REGION Network 68: **** 4.4 - Machine Status - Calculation **** Que Message Request 13 / **** 4.4 - Machine Status - Calculation **** Queue Message Request 13
   // Que Message Request 13 / Queue Message Request 13
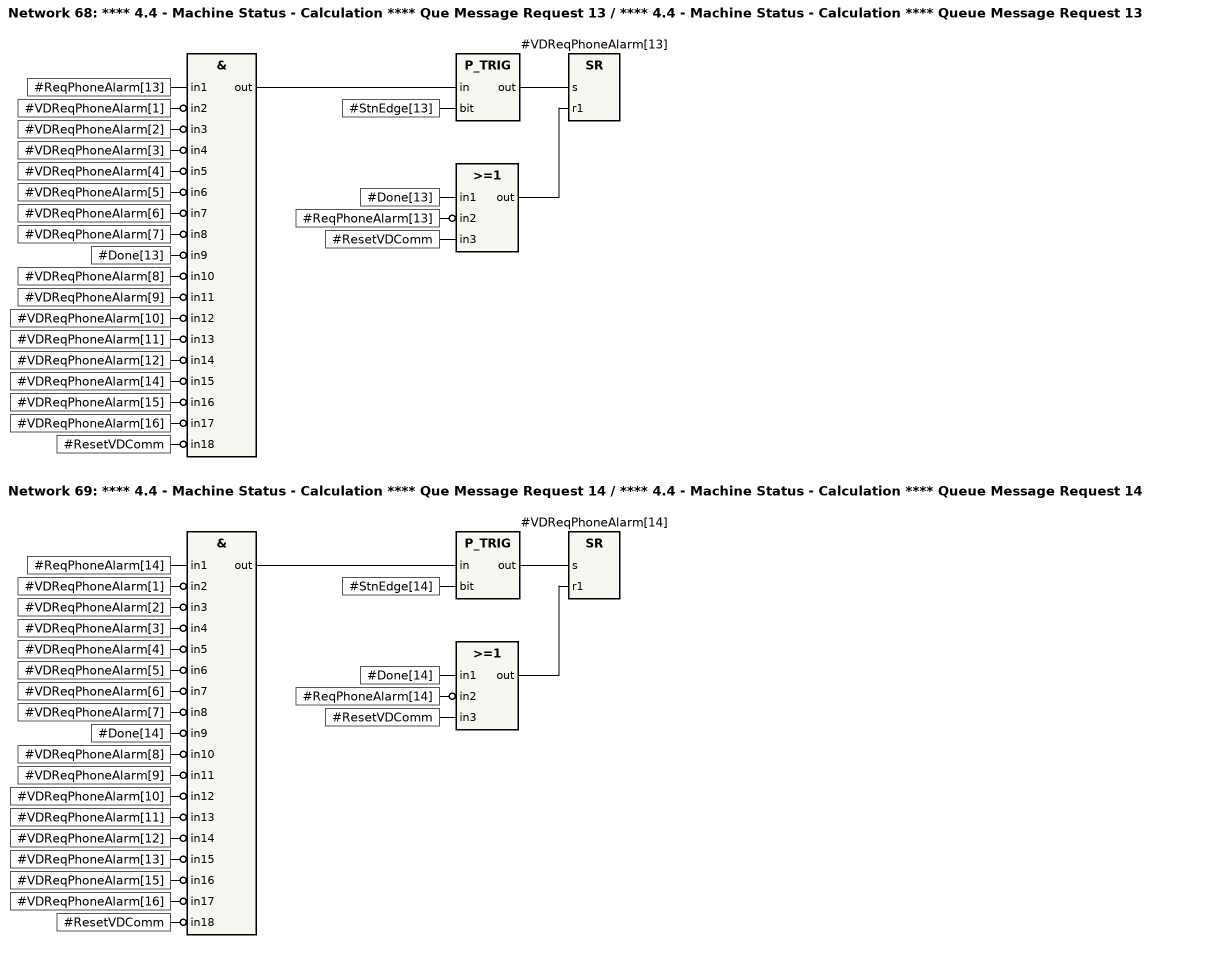
   #_w1 := #ReqPhoneAlarm[13] AND NOT #VDReqPhoneAlarm[1] AND NOT #VDReqPhoneAlarm[2] AND NOT #VDReqPhoneAlarm[3] AND NOT #VDReqPhoneAlarm[4] AND NOT #VDReqPhoneAlarm[5] AND NOT #VDReqPhoneAlarm[6] AND NOT #VDReqPhoneAlarm[7] AND NOT #Done[13] AND NOT #VDReqPhoneAlarm[8] AND NOT #VDReqPhoneAlarm[9] AND NOT #VDReqPhoneAlarm[10] AND NOT #VDReqPhoneAlarm[11] AND NOT #VDReqPhoneAlarm[12] AND NOT #VDReqPhoneAlarm[14] AND NOT #VDReqPhoneAlarm[15] AND NOT #VDReqPhoneAlarm[16] AND NOT #ResetVDComm;
   #_w2 := #_w1 AND NOT #StnEdge[13];   // rising edge
   #StnEdge[13] := #_w1;
   IF #_w2 THEN
       #VDReqPhoneAlarm[13] := TRUE;   // SR flip-flop
   END_IF;
   IF #Done[13] OR NOT #ReqPhoneAlarm[13] OR #ResetVDComm THEN #VDReqPhoneAlarm[13] := FALSE; END_IF;
END_REGION

REGION Network 69: **** 4.4 - Machine Status - Calculation **** Que Message Request 14 / **** 4.4 - Machine Status - Calculation **** Queue Message Request 14
   // Que Message Request 14 / Queue Message Request 14
   #_w1 := #ReqPhoneAlarm[14] AND NOT #VDReqPhoneAlarm[1] AND NOT #VDReqPhoneAlarm[2] AND NOT #VDReqPhoneAlarm[3] AND NOT #VDReqPhoneAlarm[4] AND NOT #VDReqPhoneAlarm[5] AND NOT #VDReqPhoneAlarm[6] AND NOT #VDReqPhoneAlarm[7] AND NOT #Done[14] AND NOT #VDReqPhoneAlarm[8] AND NOT #VDReqPhoneAlarm[9] AND NOT #VDReqPhoneAlarm[10] AND NOT #VDReqPhoneAlarm[11] AND NOT #VDReqPhoneAlarm[12] AND NOT #VDReqPhoneAlarm[13] AND NOT #VDReqPhoneAlarm[15] AND NOT #VDReqPhoneAlarm[16] AND NOT #ResetVDComm;
   #_w2 := #_w1 AND NOT #StnEdge[14];   // rising edge
   #StnEdge[14] := #_w1;
   IF #_w2 THEN
       #VDReqPhoneAlarm[14] := TRUE;   // SR flip-flop
   END_IF;
   IF #Done[14] OR NOT #ReqPhoneAlarm[14] OR #ResetVDComm THEN #VDReqPhoneAlarm[14] := FALSE; END_IF;
END_REGION

REGION Network 70: **** 4.4 - Machine Status - Calculation **** Que Message Request 15 / **** 4.4 - Machine Status - Calculation **** Queue Message Request 15
   // Que Message Request 15 / Queue Message Request 15
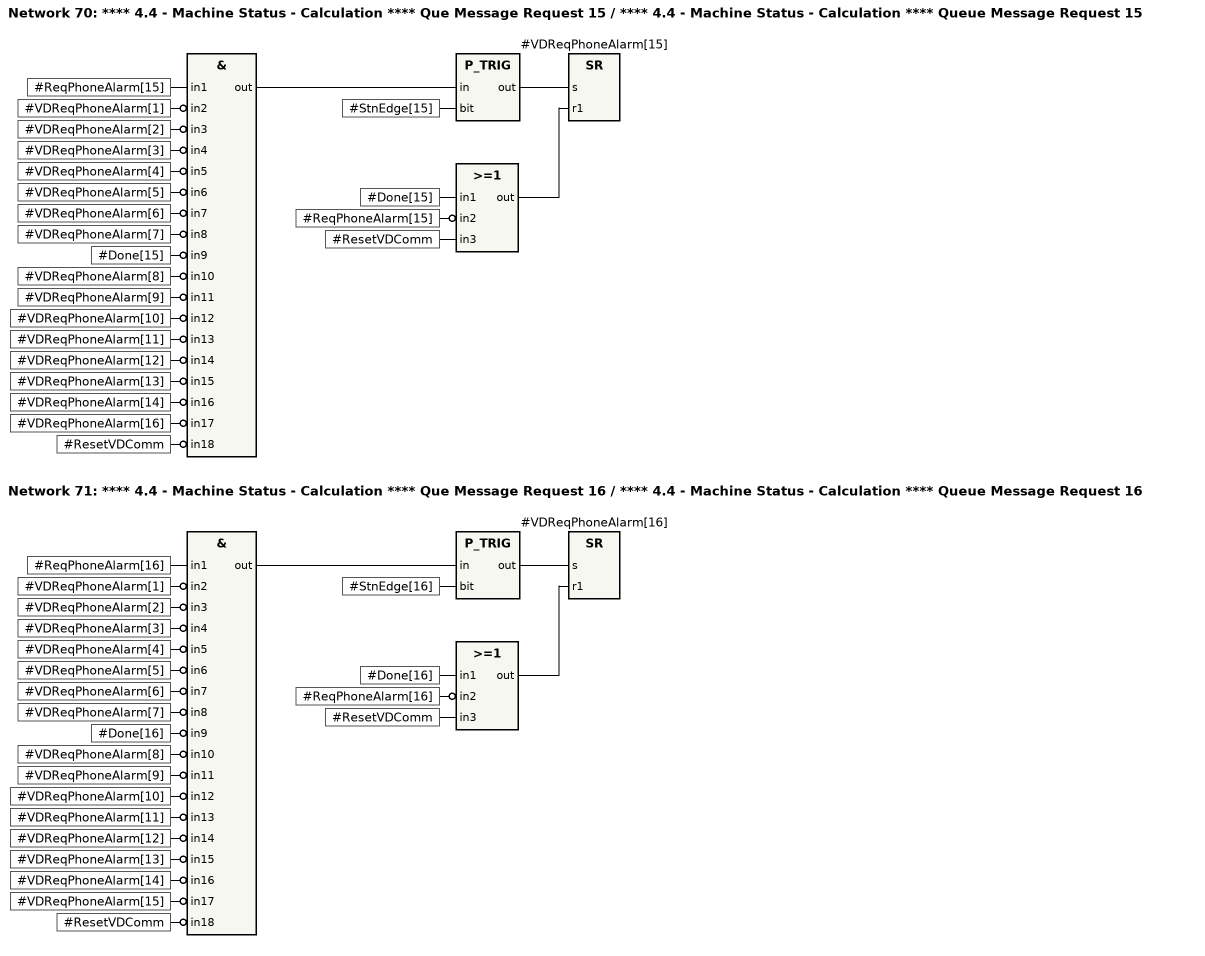
   #_w1 := #ReqPhoneAlarm[15] AND NOT #VDReqPhoneAlarm[1] AND NOT #VDReqPhoneAlarm[2] AND NOT #VDReqPhoneAlarm[3] AND NOT #VDReqPhoneAlarm[4] AND NOT #VDReqPhoneAlarm[5] AND NOT #VDReqPhoneAlarm[6] AND NOT #VDReqPhoneAlarm[7] AND NOT #Done[15] AND NOT #VDReqPhoneAlarm[8] AND NOT #VDReqPhoneAlarm[9] AND NOT #VDReqPhoneAlarm[10] AND NOT #VDReqPhoneAlarm[11] AND NOT #VDReqPhoneAlarm[12] AND NOT #VDReqPhoneAlarm[13] AND NOT #VDReqPhoneAlarm[14] AND NOT #VDReqPhoneAlarm[16] AND NOT #ResetVDComm;
   #_w2 := #_w1 AND NOT #StnEdge[15];   // rising edge
   #StnEdge[15] := #_w1;
   IF #_w2 THEN
       #VDReqPhoneAlarm[15] := TRUE;   // SR flip-flop
   END_IF;
   IF #Done[15] OR NOT #ReqPhoneAlarm[15] OR #ResetVDComm THEN #VDReqPhoneAlarm[15] := FALSE; END_IF;
END_REGION

REGION Network 71: **** 4.4 - Machine Status - Calculation **** Que Message Request 16 / **** 4.4 - Machine Status - Calculation **** Queue Message Request 16
   // Que Message Request 16 / Queue Message Request 16
   #_w1 := #ReqPhoneAlarm[16] AND NOT #VDReqPhoneAlarm[1] AND NOT #VDReqPhoneAlarm[2] AND NOT #VDReqPhoneAlarm[3] AND NOT #VDReqPhoneAlarm[4] AND NOT #VDReqPhoneAlarm[5] AND NOT #VDReqPhoneAlarm[6] AND NOT #VDReqPhoneAlarm[7] AND NOT #Done[16] AND NOT #VDReqPhoneAlarm[8] AND NOT #VDReqPhoneAlarm[9] AND NOT #VDReqPhoneAlarm[10] AND NOT #VDReqPhoneAlarm[11] AND NOT #VDReqPhoneAlarm[12] AND NOT #VDReqPhoneAlarm[13] AND NOT #VDReqPhoneAlarm[14] AND NOT #VDReqPhoneAlarm[15] AND NOT #ResetVDComm;
   #_w2 := #_w1 AND NOT #StnEdge[16];   // rising edge
   #StnEdge[16] := #_w1;
   IF #_w2 THEN
       #VDReqPhoneAlarm[16] := TRUE;   // SR flip-flop
   END_IF;
   IF #Done[16] OR NOT #ReqPhoneAlarm[16] OR #ResetVDComm THEN #VDReqPhoneAlarm[16] := FALSE; END_IF;
END_REGION

REGION Network 72: **** 4.6 - Machine status - Indication **** Animation / **** 4.6 - Machine status - Indication **** Animation SP1
   // Animation
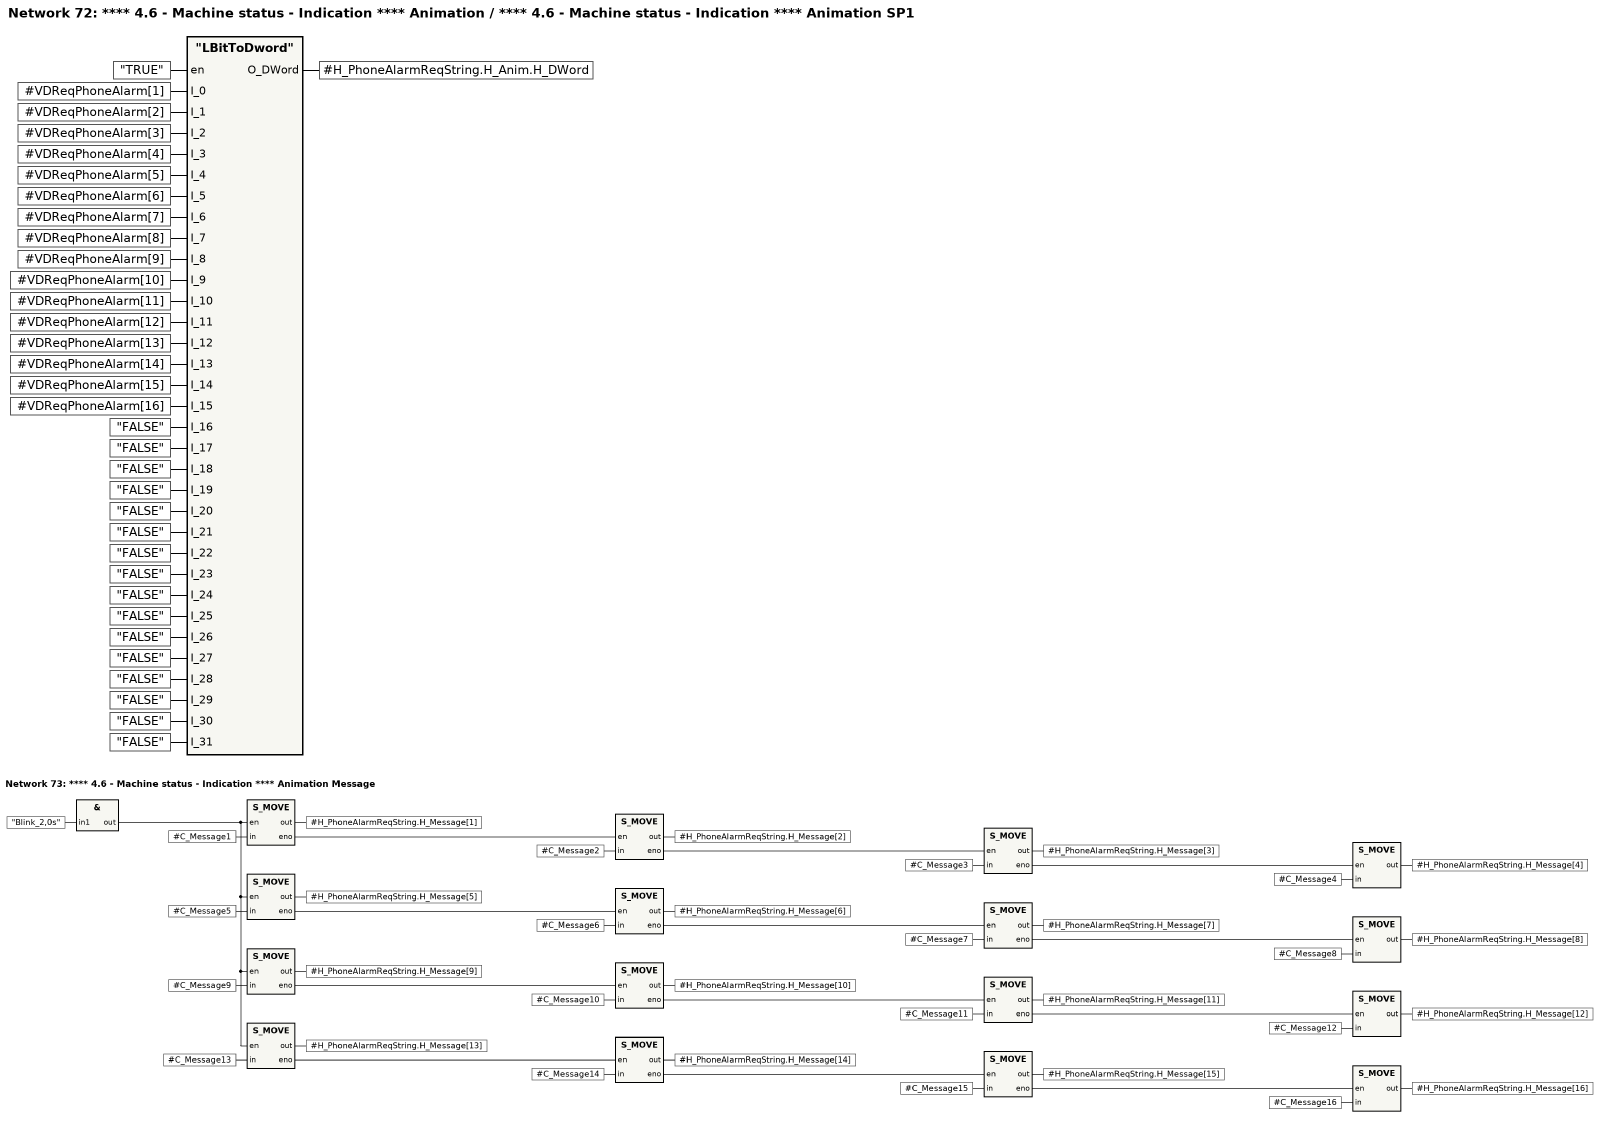
   IF "TRUE" THEN
       "LBitToDword"(I_0 := #VDReqPhoneAlarm[1],
                     I_1 := #VDReqPhoneAlarm[2],
                     I_2 := #VDReqPhoneAlarm[3],
                     I_3 := #VDReqPhoneAlarm[4],
                     I_4 := #VDReqPhoneAlarm[5],
                     I_5 := #VDReqPhoneAlarm[6],
                     I_6 := #VDReqPhoneAlarm[7],
                     I_7 := #VDReqPhoneAlarm[8],
                     I_8 := #VDReqPhoneAlarm[9],
                     I_9 := #VDReqPhoneAlarm[10],
                     I_10 := #VDReqPhoneAlarm[11],
                     I_11 := #VDReqPhoneAlarm[12],
                     I_12 := #VDReqPhoneAlarm[13],
                     I_13 := #VDReqPhoneAlarm[14],
                     I_14 := #VDReqPhoneAlarm[15],
                     I_15 := #VDReqPhoneAlarm[16],
                     I_16 := "FALSE",
                     I_17 := "FALSE",
                     I_18 := "FALSE",
                     I_19 := "FALSE",
                     I_20 := "FALSE",
                     I_21 := "FALSE",
                     I_22 := "FALSE",
                     I_23 := "FALSE",
                     I_24 := "FALSE",
                     I_25 := "FALSE",
                     I_26 := "FALSE",
                     I_27 := "FALSE",
                     I_28 := "FALSE",
                     I_29 := "FALSE",
                     I_30 := "FALSE",
                     I_31 := "FALSE",
                     O_DWord => #H_PhoneAlarmReqString.H_Anim.H_DWord);
   END_IF;
END_REGION

REGION Network 73: **** 4.6 - Machine status - Indication **** Animation Message
   IF "Blink_2,0s" THEN
       #H_PhoneAlarmReqString.H_Message[1] := #C_Message1;
       #H_PhoneAlarmReqString.H_Message[2] := #C_Message2;
       #H_PhoneAlarmReqString.H_Message[3] := #C_Message3;
       #H_PhoneAlarmReqString.H_Message[4] := #C_Message4;
       #H_PhoneAlarmReqString.H_Message[5] := #C_Message5;
       #H_PhoneAlarmReqString.H_Message[6] := #C_Message6;
       #H_PhoneAlarmReqString.H_Message[7] := #C_Message7;
       #H_PhoneAlarmReqString.H_Message[8] := #C_Message8;
       #H_PhoneAlarmReqString.H_Message[9] := #C_Message9;
       #H_PhoneAlarmReqString.H_Message[10] := #C_Message10;
       #H_PhoneAlarmReqString.H_Message[11] := #C_Message11;
       #H_PhoneAlarmReqString.H_Message[12] := #C_Message12;
       #H_PhoneAlarmReqString.H_Message[13] := #C_Message13;
       #H_PhoneAlarmReqString.H_Message[14] := #C_Message14;
       #H_PhoneAlarmReqString.H_Message[15] := #C_Message15;
       #H_PhoneAlarmReqString.H_Message[16] := #C_Message16;
   END_IF;
END_REGION

REGION Network 74: **** 4.6 - Machine status - Indication **** Animation Message Type
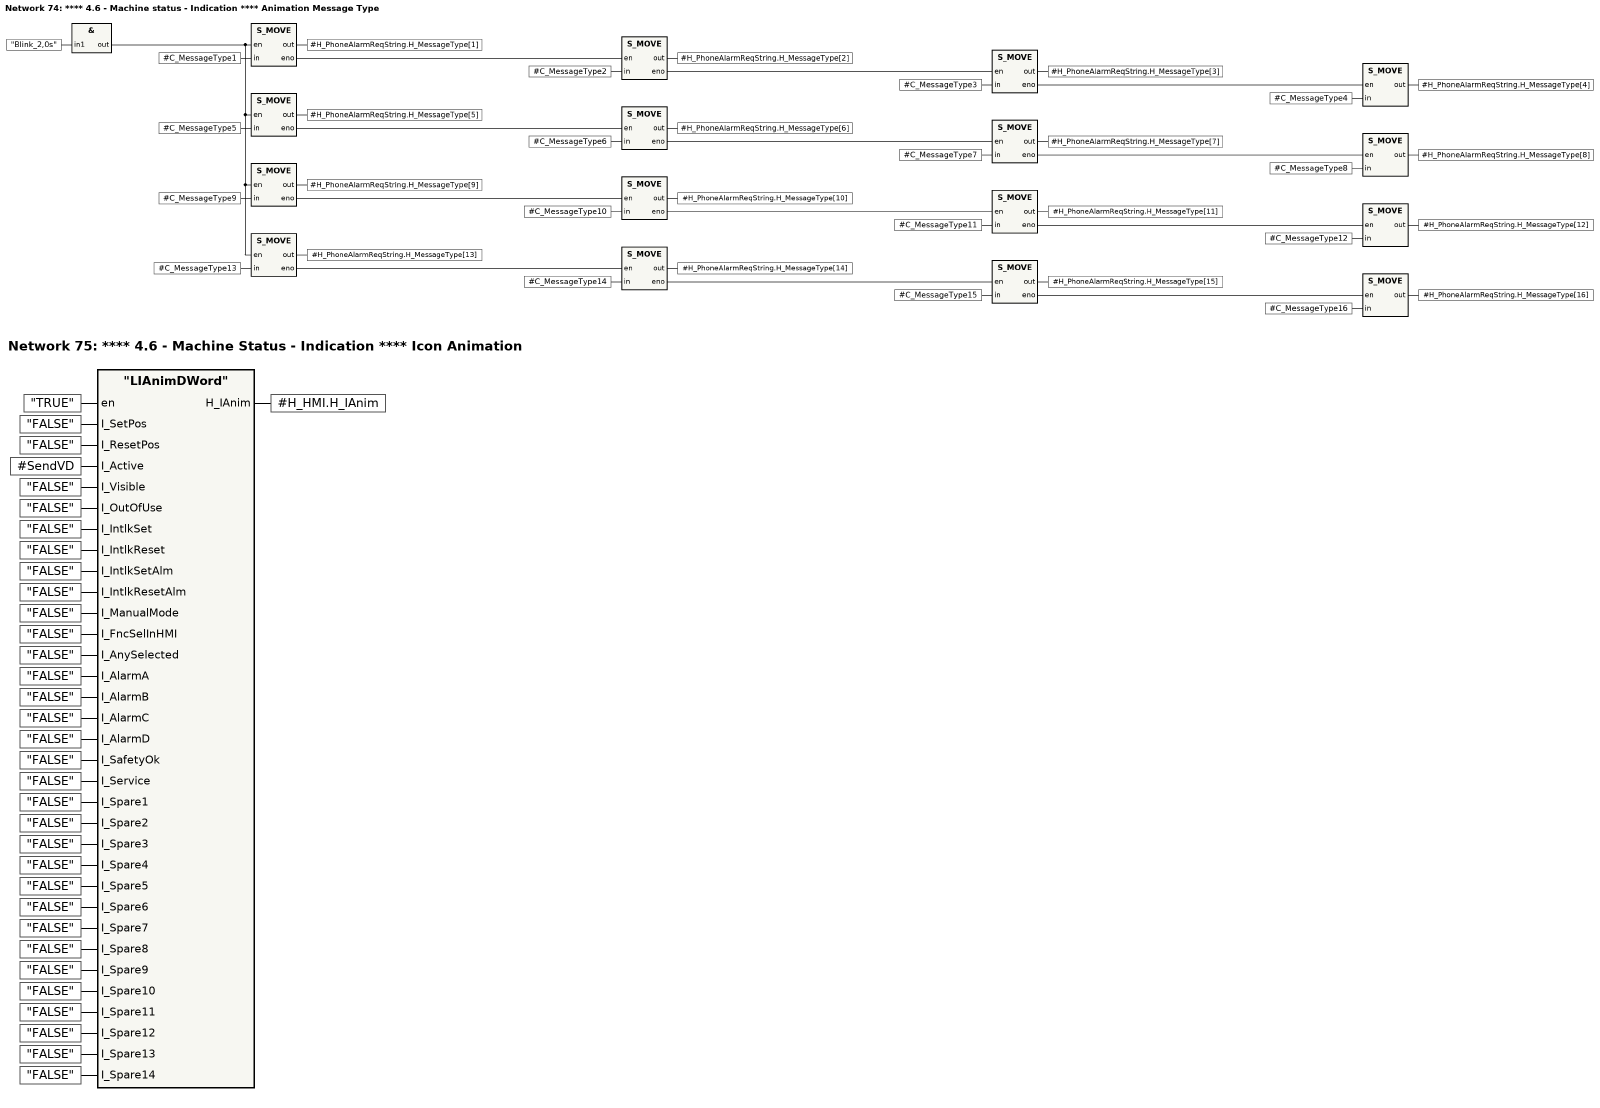
   IF "Blink_2,0s" THEN
       #H_PhoneAlarmReqString.H_MessageType[1] := #C_MessageType1;
       #H_PhoneAlarmReqString.H_MessageType[2] := #C_MessageType2;
       #H_PhoneAlarmReqString.H_MessageType[3] := #C_MessageType3;
       #H_PhoneAlarmReqString.H_MessageType[4] := #C_MessageType4;
       #H_PhoneAlarmReqString.H_MessageType[5] := #C_MessageType5;
       #H_PhoneAlarmReqString.H_MessageType[6] := #C_MessageType6;
       #H_PhoneAlarmReqString.H_MessageType[7] := #C_MessageType7;
       #H_PhoneAlarmReqString.H_MessageType[8] := #C_MessageType8;
       #H_PhoneAlarmReqString.H_MessageType[9] := #C_MessageType9;
       #H_PhoneAlarmReqString.H_MessageType[10] := #C_MessageType10;
       #H_PhoneAlarmReqString.H_MessageType[11] := #C_MessageType11;
       #H_PhoneAlarmReqString.H_MessageType[12] := #C_MessageType12;
       #H_PhoneAlarmReqString.H_MessageType[13] := #C_MessageType13;
       #H_PhoneAlarmReqString.H_MessageType[14] := #C_MessageType14;
       #H_PhoneAlarmReqString.H_MessageType[15] := #C_MessageType15;
       #H_PhoneAlarmReqString.H_MessageType[16] := #C_MessageType16;
   END_IF;
END_REGION

REGION Network 75: **** 4.6 - Machine Status - Indication **** Icon Animation
   // Icon Animation
   IF "TRUE" THEN
       "LIAnimDWord"(I_SetPos := "FALSE",
                     I_ResetPos := "FALSE",
                     I_Active := #SendVD,
                     I_Visible := "FALSE",
                     I_OutOfUse := "FALSE",
                     I_IntlkSet := "FALSE",
                     I_IntlkReset := "FALSE",
                     I_IntlkSetAlm := "FALSE",
                     I_IntlkResetAlm := "FALSE",
                     I_ManualMode := "FALSE",
                     I_FncSelInHMI := "FALSE",
                     I_AnySelected := "FALSE",
                     I_AlarmA := "FALSE",
                     I_AlarmB := "FALSE",
                     I_AlarmC := "FALSE",
                     I_AlarmD := "FALSE",
                     I_SafetyOk := "FALSE",
                     I_Service := "FALSE",
                     I_Spare1 := "FALSE",
                     I_Spare2 := "FALSE",
                     I_Spare3 := "FALSE",
                     I_Spare4 := "FALSE",
                     I_Spare5 := "FALSE",
                     I_Spare6 := "FALSE",
                     I_Spare7 := "FALSE",
                     I_Spare8 := "FALSE",
                     I_Spare9 := "FALSE",
                     I_Spare10 := "FALSE",
                     I_Spare11 := "FALSE",
                     I_Spare12 := "FALSE",
                     I_Spare13 := "FALSE",
                     I_Spare14 := "FALSE",
                     H_IAnim => #H_HMI.H_IAnim);
   END_IF;
END_REGION

REGION Network 76: **** 8 - Outputs **** Data / **** 8 - Outputs **** Prepare Data
   // Data / Prepare Data
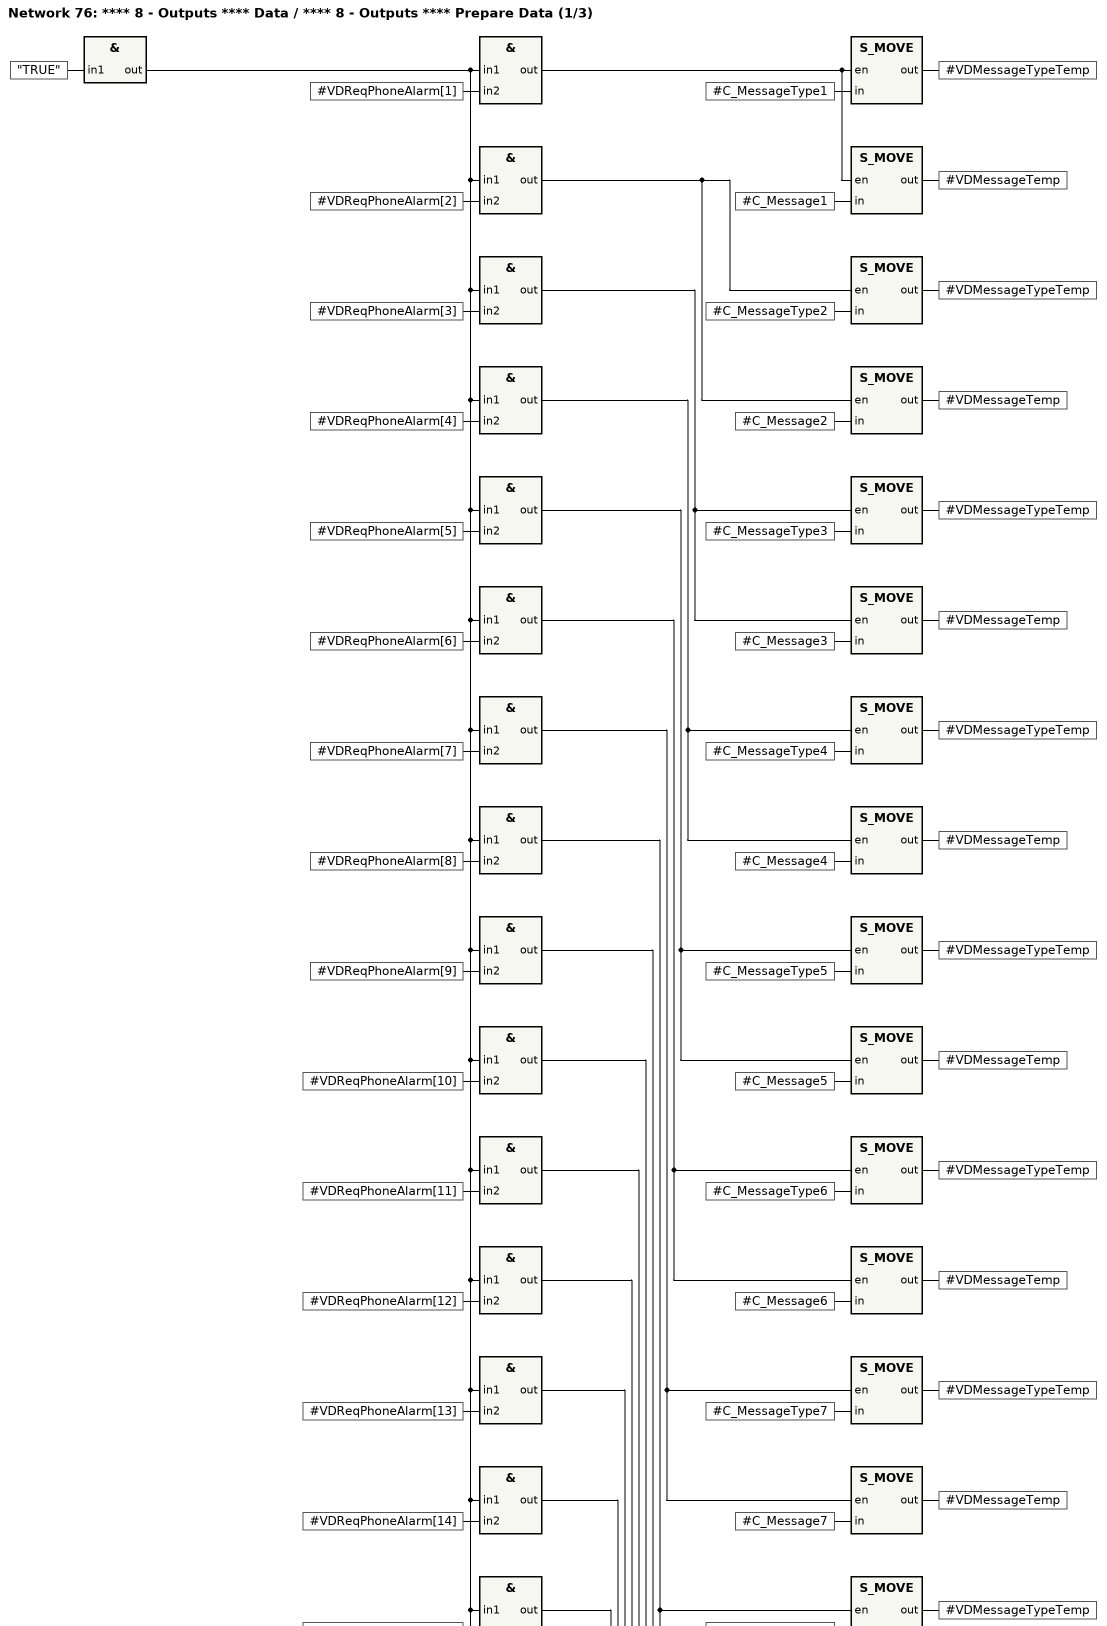
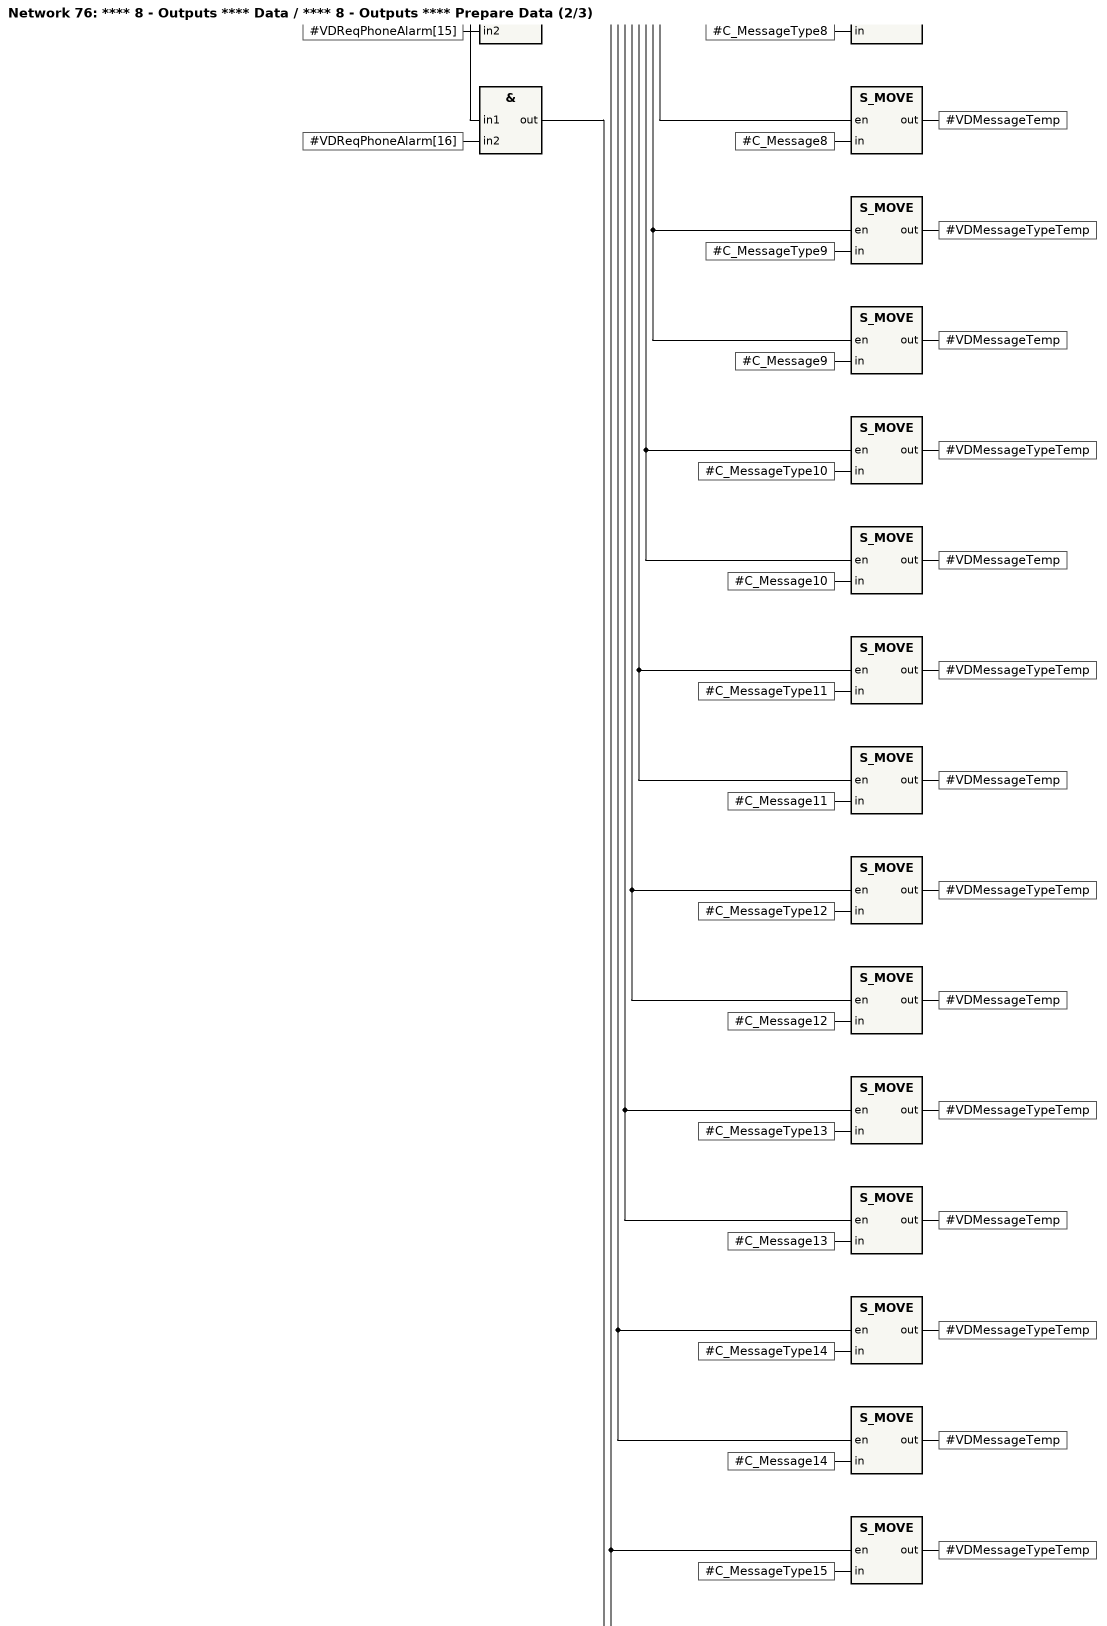
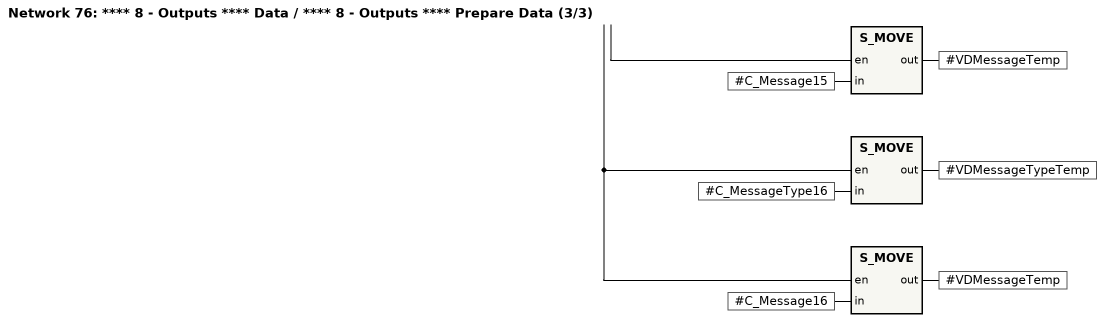
   IF "TRUE" AND #VDReqPhoneAlarm[1] THEN
       #VDMessageTypeTemp := #C_MessageType1;
       #VDMessageTemp := #C_Message1;
   END_IF;
   IF "TRUE" AND #VDReqPhoneAlarm[2] THEN
       #VDMessageTypeTemp := #C_MessageType2;
       #VDMessageTemp := #C_Message2;
   END_IF;
   IF "TRUE" AND #VDReqPhoneAlarm[3] THEN
       #VDMessageTypeTemp := #C_MessageType3;
       #VDMessageTemp := #C_Message3;
   END_IF;
   IF "TRUE" AND #VDReqPhoneAlarm[4] THEN
       #VDMessageTypeTemp := #C_MessageType4;
       #VDMessageTemp := #C_Message4;
   END_IF;
   IF "TRUE" AND #VDReqPhoneAlarm[5] THEN
       #VDMessageTypeTemp := #C_MessageType5;
       #VDMessageTemp := #C_Message5;
   END_IF;
   IF "TRUE" AND #VDReqPhoneAlarm[6] THEN
       #VDMessageTypeTemp := #C_MessageType6;
       #VDMessageTemp := #C_Message6;
   END_IF;
   IF "TRUE" AND #VDReqPhoneAlarm[7] THEN
       #VDMessageTypeTemp := #C_MessageType7;
       #VDMessageTemp := #C_Message7;
   END_IF;
   IF "TRUE" AND #VDReqPhoneAlarm[8] THEN
       #VDMessageTypeTemp := #C_MessageType8;
       #VDMessageTemp := #C_Message8;
   END_IF;
   IF "TRUE" AND #VDReqPhoneAlarm[9] THEN
       #VDMessageTypeTemp := #C_MessageType9;
       #VDMessageTemp := #C_Message9;
   END_IF;
   IF "TRUE" AND #VDReqPhoneAlarm[10] THEN
       #VDMessageTypeTemp := #C_MessageType10;
       #VDMessageTemp := #C_Message10;
   END_IF;
   IF "TRUE" AND #VDReqPhoneAlarm[11] THEN
       #VDMessageTypeTemp := #C_MessageType11;
       #VDMessageTemp := #C_Message11;
   END_IF;
   IF "TRUE" AND #VDReqPhoneAlarm[12] THEN
       #VDMessageTypeTemp := #C_MessageType12;
       #VDMessageTemp := #C_Message12;
   END_IF;
   IF "TRUE" AND #VDReqPhoneAlarm[13] THEN
       #VDMessageTypeTemp := #C_MessageType13;
       #VDMessageTemp := #C_Message13;
   END_IF;
   IF "TRUE" AND #VDReqPhoneAlarm[14] THEN
       #VDMessageTypeTemp := #C_MessageType14;
       #VDMessageTemp := #C_Message14;
   END_IF;
   IF "TRUE" AND #VDReqPhoneAlarm[15] THEN
       #VDMessageTypeTemp := #C_MessageType15;
       #VDMessageTemp := #C_Message15;
   END_IF;
   IF "TRUE" AND #VDReqPhoneAlarm[16] THEN
       #VDMessageTypeTemp := #C_MessageType16;
       #VDMessageTemp := #C_Message16;
   END_IF;
END_REGION

REGION Network 77: **** 8 - Outputs **** Prepare MessageType and Message
   // Prepare Message
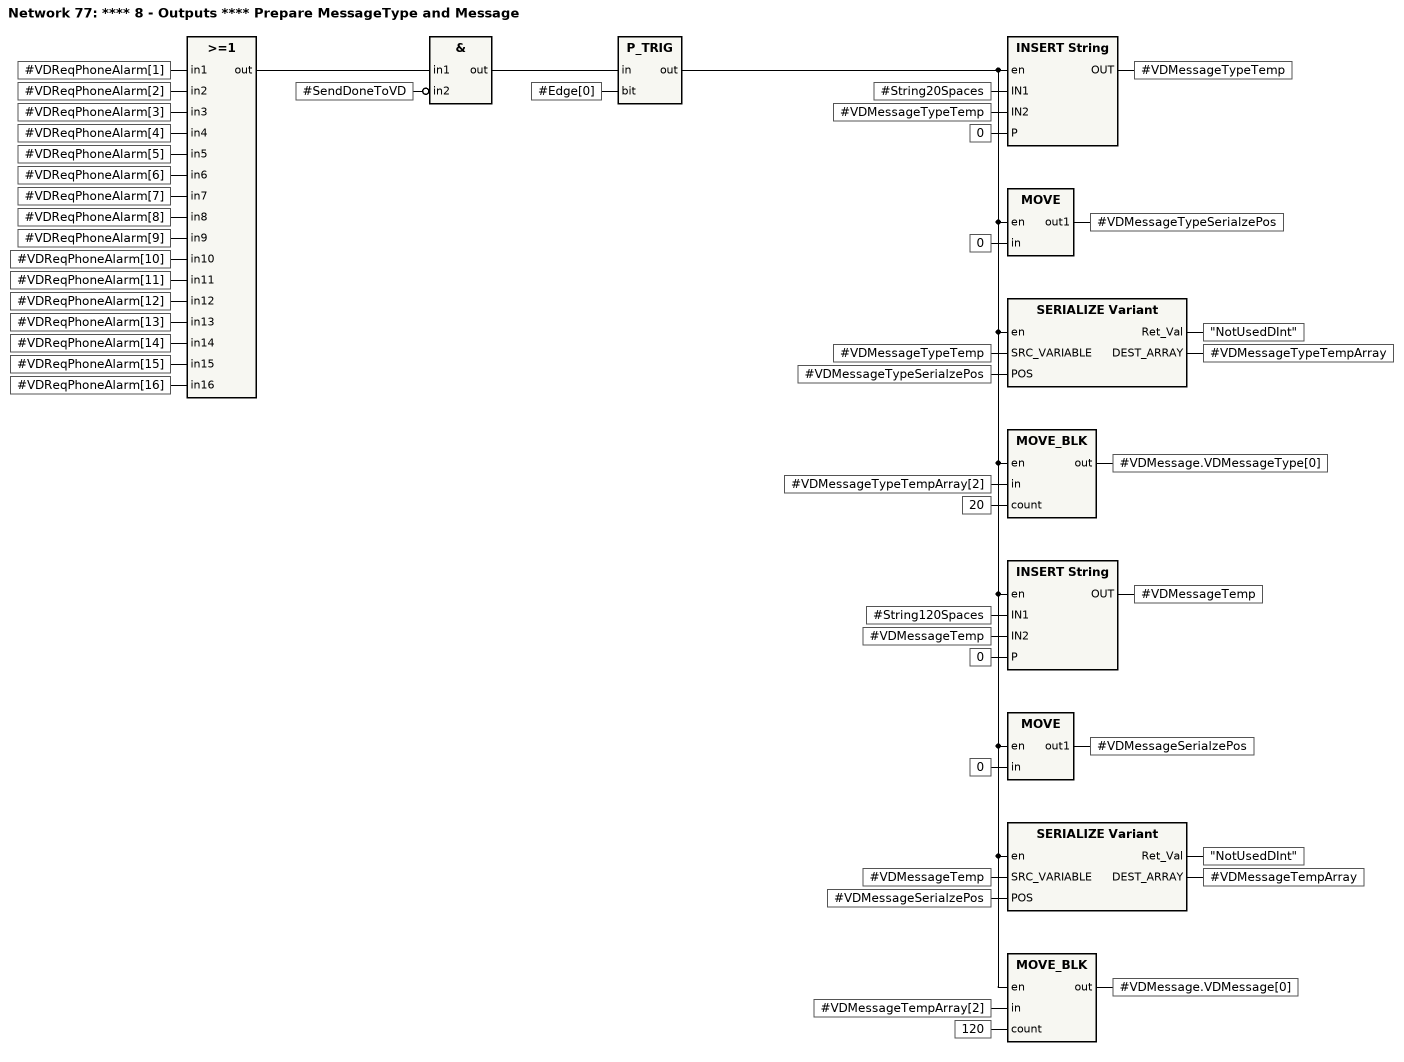
   #_w1 := (#VDReqPhoneAlarm[1] OR #VDReqPhoneAlarm[2] OR #VDReqPhoneAlarm[3] OR #VDReqPhoneAlarm[4] OR #VDReqPhoneAlarm[5] OR #VDReqPhoneAlarm[6] OR #VDReqPhoneAlarm[7] OR #VDReqPhoneAlarm[8] OR #VDReqPhoneAlarm[9] OR #VDReqPhoneAlarm[10] OR #VDReqPhoneAlarm[11] OR #VDReqPhoneAlarm[12] OR #VDReqPhoneAlarm[13] OR #VDReqPhoneAlarm[14] OR #VDReqPhoneAlarm[15] OR #VDReqPhoneAlarm[16]) AND NOT #SendDoneToVD;
   #_w2 := #_w1 AND NOT #Edge[0];   // rising edge
   #Edge[0] := #_w1;
   IF #_w2 THEN
       INSERT(IN1 := #String20Spaces, IN2 := #VDMessageTypeTemp, P := 0, OUT => #VDMessageTypeTemp);
       #VDMessageTypeSerialzePos := 0;
       "NotUsedDInt" := Serialize(SRC_VARIABLE := #VDMessageTypeTemp,
                               POS := #VDMessageTypeSerialzePos,
                               DEST_ARRAY => #VDMessageTypeTempArray);
       MOVE_BLK(IN := #VDMessageTypeTempArray[2], COUNT := 20, OUT => #VDMessage.VDMessageType[0]);
       INSERT(IN1 := #String120Spaces, IN2 := #VDMessageTemp, P := 0, OUT => #VDMessageTemp);
       #VDMessageSerialzePos := 0;
       "NotUsedDInt" := Serialize(SRC_VARIABLE := #VDMessageTemp,
                               POS := #VDMessageSerialzePos,
                               DEST_ARRAY => #VDMessageTempArray);
       MOVE_BLK(IN := #VDMessageTempArray[2], COUNT := 120, OUT => #VDMessage.VDMessage[0]);
   END_IF;
END_REGION

REGION Network 78: **** 8 - Outputs **** Send To VD
   // Send To VD
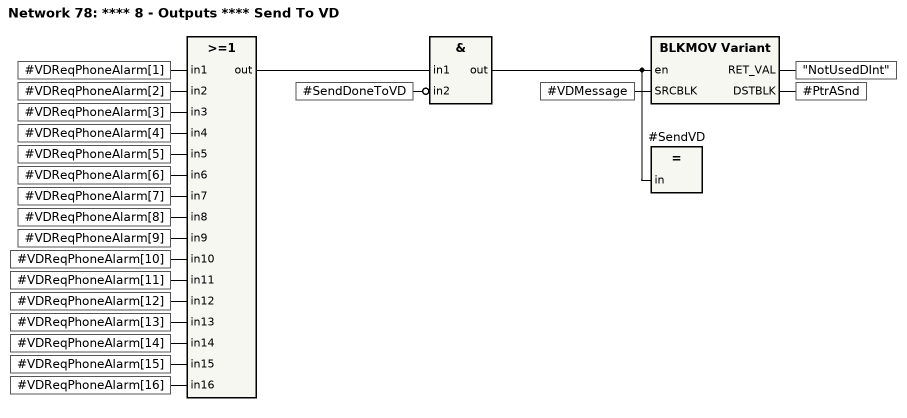
   #_w1 := (#VDReqPhoneAlarm[1] OR #VDReqPhoneAlarm[2] OR #VDReqPhoneAlarm[3] OR #VDReqPhoneAlarm[4] OR #VDReqPhoneAlarm[5] OR #VDReqPhoneAlarm[6] OR #VDReqPhoneAlarm[7] OR #VDReqPhoneAlarm[8] OR #VDReqPhoneAlarm[9] OR #VDReqPhoneAlarm[10] OR #VDReqPhoneAlarm[11] OR #VDReqPhoneAlarm[12] OR #VDReqPhoneAlarm[13] OR #VDReqPhoneAlarm[14] OR #VDReqPhoneAlarm[15] OR #VDReqPhoneAlarm[16]) AND NOT #SendDoneToVD;
   IF #_w1 THEN "NotUsedDInt" := BLKMOV(SRCBLK := #VDMessage, DSTBLK => #PtrASnd); END_IF;
   #SendVD := #_w1;
END_REGION
END_FUNCTION_BLOCK

FUNCTION_BLOCK "209210NCB01TagSeq"   // FB340, GRAPH
{ S7_Optimized_Access := 'TRUE' }
VERSION : 0.1
// stored: AcknowledgeErrorsRequired true, AutoNumber false, GraphVersion 6.0, InitialValuesAcquisition false, IsIECCheckEnabled false, LanguageInNetworks FBD, LockOperatingMode false, PermanentILProcessingInMANMode false, SetENOAutomatically false, SkipSteps false, UDAEnableTagReadback false, WithAlarmHandling true
   // inherited from GRAPH_BASE
   VAR
      OFF_SQ_BASE : Bool;
   END_VAR
   VAR_INPUT
      OFF_SQ { ExternalWritable := 'False'} : Bool := false;   // Turn sequence off
      INIT_SQ { ExternalWritable := 'False'} : Bool := false;   // Set sequence to initial state
      ACK_EF { ExternalWritable := 'False'} : Bool := false;   // Acknowledge all errors and faults
      S_PREV { ExternalWritable := 'False'} : Bool := false;   // Output previous step in parameter S_NO
      S_NEXT { ExternalWritable := 'False'} : Bool := false;   // Indicate next step in parameter S_NO
      SW_AUTO { ExternalWritable := 'False'} : Bool := false;   // Automatic mode
      SW_TAP { ExternalWritable := 'False'} : Bool := false;   // Semiautomatic/switch with transition
      SW_TOP { ExternalWritable := 'False'} : Bool := false;   // Semiautomatic/ignore transition
      SW_MAN { ExternalWritable := 'False'} : Bool := false;   // Manual mode
      S_SEL { ExternalWritable := 'False'} : Int := 0;   // Select step to be output to S_NO
      S_ON { ExternalWritable := 'False'} : Bool := false;   // Activate step indicated in S_NO
      S_OFF { ExternalWritable := 'False'} : Bool := false;   // Deactivate step indicated S_NO
      T_PUSH { ExternalWritable := 'False'} : Bool := false;   // Enable transition to switch in semi automatic mode
   END_VAR
   VAR_OUTPUT
      S_NO { ExternalWritable := 'False'} : Int := 0;   // Step number
      S_MORE { ExternalWritable := 'False'} : Bool := false;   // More steps are available and can be shown in S_NO
      S_ACTIVE { ExternalWritable := 'False'} : Bool := false;   // Step indicated in S_NO is active
      ERR_FLT { ExternalWritable := 'False'} : Bool := false;   // Interlock or supervision group error
      AUTO_ON { ExternalWritable := 'False'} : Bool := false;   // Automatic mode is active
      TAP_ON { ExternalWritable := 'False'} : Bool := false;   // Semiautomatic mode/step with transition enabled
      TOP_ON { ExternalWritable := 'False'} : Bool := false;   // Semiautomatic mode/ignore transition enabled
      MAN_ON { ExternalWritable := 'False'} : Bool := false;   // Manual mode is active
   END_VAR
BEGIN
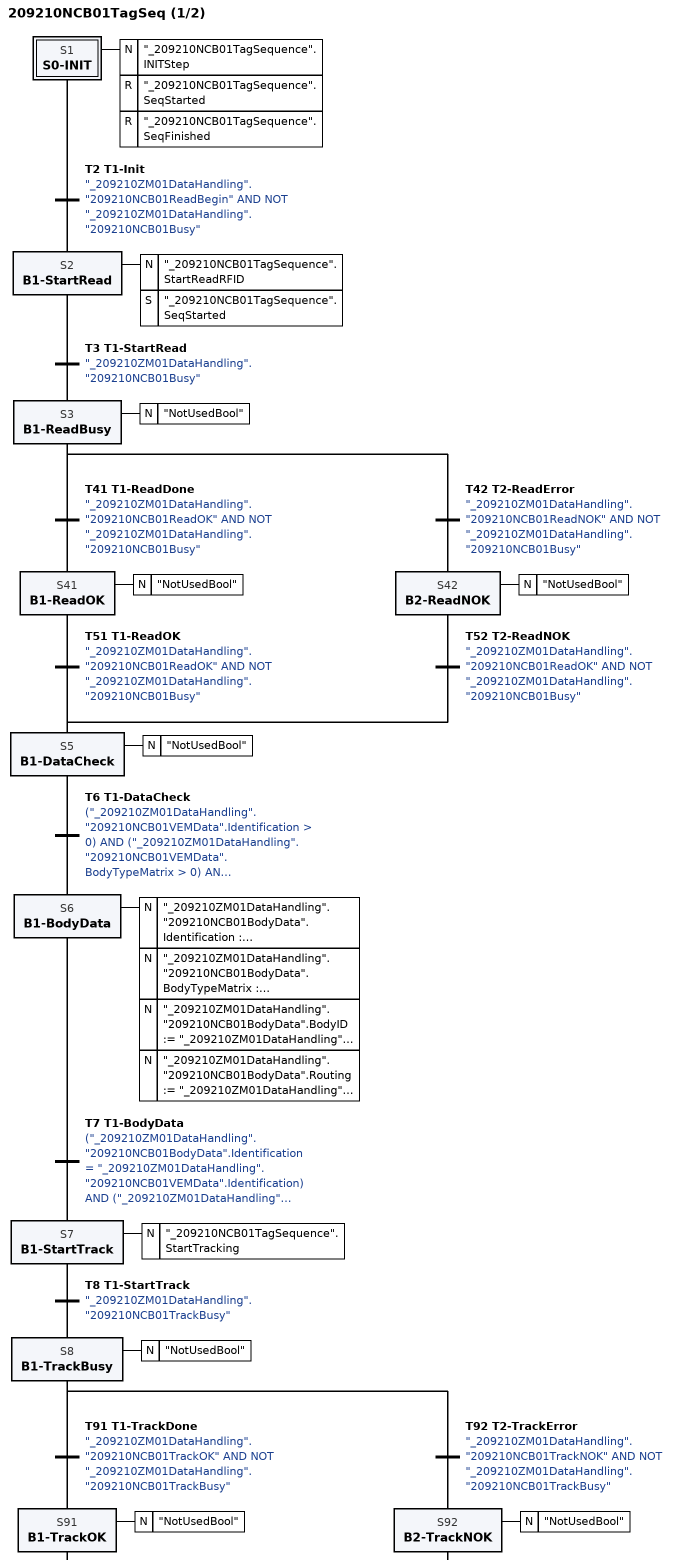
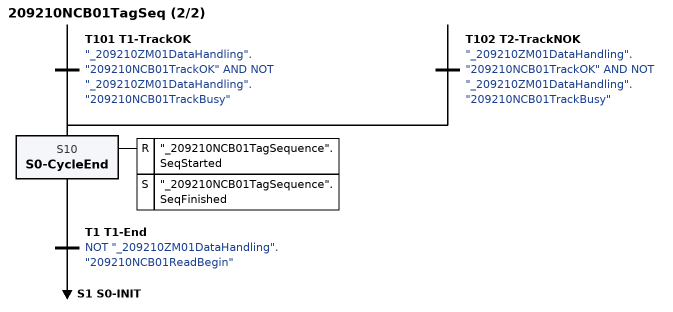
   // sequencer 1: 209210NCB01 Tag Sequence
   // Tag Sequence of 209210NCB01
   INITIAL_STEP "S0-INIT":   // S1, max time T#10S, warning time T#7S
      interlock C := (none);   // Not used
      supervision V := (none);   // Not Used
      // INIT
              N    "_209210NCB01TagSequence".INITStep
              R    "_209210NCB01TagSequence".SeqStarted
              R    "_209210NCB01TagSequence".SeqFinished
   END_STEP
   TRANSITION "T1-Init" FROM "S0-INIT" TO "B1-StartRead"   // T2
      := "_209210ZM01DataHandling"."209210NCB01ReadBegin" AND NOT "_209210ZM01DataHandling"."209210NCB01Busy";
   END_TRANSITION
   STEP "B1-StartRead":   // S2, max time T#10S, warning time T#7S
      interlock C := (none);   // Not Used
      supervision V := (none);   // Not Used
      // Start Getting VEM Data by Reading the Tag with RFID
              N    "_209210NCB01TagSequence".StartReadRFID
              S    "_209210NCB01TagSequence".SeqStarted
   END_STEP
   TRANSITION "T1-StartRead" FROM "B1-StartRead" TO "B1-ReadBusy"   // T3
      := "_209210ZM01DataHandling"."209210NCB01Busy";
   END_TRANSITION
   STEP "B1-ReadBusy":   // S3, max time T#10S, warning time T#7S
      interlock C := (none);   // Not Used
      supervision V := (none);   // Not Used
      // The Tag Reading is Busy
              N    "NotUsedBool"
   END_STEP
   TRANSITION "T1-ReadDone" FROM "B1-ReadBusy" TO "B1-ReadOK"   // T41
      := "_209210ZM01DataHandling"."209210NCB01ReadOK" AND NOT "_209210ZM01DataHandling"."209210NCB01Busy";
   END_TRANSITION
   TRANSITION "T2-ReadError" FROM "B1-ReadBusy" TO "B2-ReadNOK"   // T42
      := "_209210ZM01DataHandling"."209210NCB01ReadNOK" AND NOT "_209210ZM01DataHandling"."209210NCB01Busy";
   END_TRANSITION
   STEP "B1-ReadOK":   // S41, max time T#10S, warning time T#7S
      interlock C := (none);   // Not Used
      supervision V := (none);   // Not Used
      // Reading of Tag is OK
              N    "NotUsedBool"
   END_STEP
   TRANSITION "T1-ReadOK" FROM "B1-ReadOK" TO "B1-DataCheck"   // T51
      := "_209210ZM01DataHandling"."209210NCB01ReadOK" AND NOT "_209210ZM01DataHandling"."209210NCB01Busy";
   END_TRANSITION
   STEP "B2-ReadNOK":   // S42, max time T#10S, warning time T#7S
      interlock C := (none);   // Not Used
      supervision V := (none);   // Not Used
      // Reading of Tag is Not OK
              N    "NotUsedBool"
   END_STEP
   TRANSITION "T2-ReadNOK" FROM "B2-ReadNOK" TO "B1-DataCheck"   // T52
      := "_209210ZM01DataHandling"."209210NCB01ReadOK" AND NOT "_209210ZM01DataHandling"."209210NCB01Busy";
   END_TRANSITION
   STEP "S0-CycleEnd":   // S10, max time T#10S, warning time T#7S
      interlock C := (none);   // Not Used
      supervision V := (none);   // Not Used
      // Finished
              R    "_209210NCB01TagSequence".SeqStarted
              S    "_209210NCB01TagSequence".SeqFinished
   END_STEP
   TRANSITION "T1-End" FROM "S0-CycleEnd" TO "S0-INIT"   // T1, jump
      := NOT "_209210ZM01DataHandling"."209210NCB01ReadBegin";
   END_TRANSITION
   STEP "B1-DataCheck":   // S5, max time T#10S, warning time T#7S
      interlock C := (none);   // Not Used
      supervision V := (none);   // Not Used
      // Check if the Received Data is Valid
              N    "NotUsedBool"
   END_STEP
   TRANSITION "T1-DataCheck" FROM "B1-DataCheck" TO "B1-BodyData"   // T6
      := ("_209210ZM01DataHandling"."209210NCB01VEMData".Identification > 0) AND ("_209210ZM01DataHandling"."209210NCB01VEMData".BodyTypeMatrix > 0) AND ("_209210ZM01DataHandling"."209210NCB01VEMData".BodyID > 0) AND ("_209210ZM01DataHandling"."209210NCB01VEMData".BodyID <= 9999999) AND "_209210ZM01DataHandling"."209210NCB01VEMDataValid";
   END_TRANSITION
   STEP "B1-BodyData":   // S6, max time T#10S, warning time T#7S
      interlock C := (none);   // Not Used
      supervision V := (none);   // Not Used
      // Prepare Data for local use (ex. Shift Register)
              N    "_209210ZM01DataHandling"."209210NCB01BodyData".Identification := "_209210ZM01DataHandling"."209210NCB01VEMData".Identification
              N    "_209210ZM01DataHandling"."209210NCB01BodyData".BodyTypeMatrix := "_209210ZM01DataHandling"."209210NCB01VEMData".BodyTypeMatrix
              N    "_209210ZM01DataHandling"."209210NCB01BodyData".BodyID := "_209210ZM01DataHandling"."209210NCB01VEMData".BodyID
              N    "_209210ZM01DataHandling"."209210NCB01BodyData".Routing := "_209210ZM01DataHandling"."209210NCB01VEMData".Routing
   END_STEP
   TRANSITION "T1-BodyData" FROM "B1-BodyData" TO "B1-StartTrack"   // T7
      := ("_209210ZM01DataHandling"."209210NCB01BodyData".Identification = "_209210ZM01DataHandling"."209210NCB01VEMData".Identification) AND ("_209210ZM01DataHandling"."209210NCB01BodyData".BodyTypeMatrix = "_209210ZM01DataHandling"."209210NCB01VEMData".BodyTypeMatrix) AND ("_209210ZM01DataHandling"."209210NCB01BodyData".BodyID = "_209210ZM01DataHandling"."209210NCB01VEMData".BodyID) AND ("_209210ZM01DataHandling"."209210NCB01BodyData".Routing = "_209210ZM01DataHandling"."209210NCB01VEMData".Routing);
   END_TRANSITION
   STEP "B1-StartTrack":   // S7, max time T#10S, warning time T#7S
      interlock C := (none);   // Not Used
      supervision V := (none);   // Not Used
      // Start Tracking the Body
              N    "_209210NCB01TagSequence".StartTracking
   END_STEP
   TRANSITION "T1-StartTrack" FROM "B1-StartTrack" TO "B1-TrackBusy"   // T8
      := "_209210ZM01DataHandling"."209210NCB01TrackBusy";
   END_TRANSITION
   STEP "B1-TrackOK":   // S91, max time T#10S, warning time T#7S
      interlock C := (none);   // Not Used
      supervision V := (none);   // Not Used
      // Tracking of the Body is OK
              N    "NotUsedBool"
   END_STEP
   TRANSITION "T1-TrackOK" FROM "B1-TrackOK" TO "S0-CycleEnd"   // T101
      := "_209210ZM01DataHandling"."209210NCB01TrackOK" AND NOT "_209210ZM01DataHandling"."209210NCB01TrackBusy";
   END_TRANSITION
   STEP "B2-TrackNOK":   // S92, max time T#10S, warning time T#7S
      interlock C := (none);   // Not Used
      supervision V := (none);   // Not Used
      // Tracking of the Body is Not OK
              N    "NotUsedBool"
   END_STEP
   TRANSITION "T2-TrackNOK" FROM "B2-TrackNOK" TO "S0-CycleEnd"   // T102
      := "_209210ZM01DataHandling"."209210NCB01TrackOK" AND NOT "_209210ZM01DataHandling"."209210NCB01TrackBusy";
   END_TRANSITION
   STEP "B1-TrackBusy":   // S8, max time T#10S, warning time T#7S
      interlock C := (none);   // Not Used
      supervision V := (none);   // Not Used
      // The Body Tracking is Busy
              N    "NotUsedBool"
   END_STEP
   TRANSITION "T1-TrackDone" FROM "B1-TrackBusy" TO "B1-TrackOK"   // T91
      := "_209210ZM01DataHandling"."209210NCB01TrackOK" AND NOT "_209210ZM01DataHandling"."209210NCB01TrackBusy";
   END_TRANSITION
   TRANSITION "T2-TrackError" FROM "B1-TrackBusy" TO "B2-TrackNOK"   // T92
      := "_209210ZM01DataHandling"."209210NCB01TrackNOK" AND NOT "_209210ZM01DataHandling"."209210NCB01TrackBusy";
   END_TRANSITION

   // permanent post-instructions: Not Used
END_FUNCTION_BLOCK

FUNCTION_BLOCK "209210NCB02TagSeq"   // FB341, GRAPH
{ S7_Optimized_Access := 'TRUE' }
VERSION : 0.1
// stored: AcknowledgeErrorsRequired true, AutoNumber false, GraphVersion 6.0, InitialValuesAcquisition false, IsIECCheckEnabled false, LanguageInNetworks FBD, LockOperatingMode false, PermanentILProcessingInMANMode false, SetENOAutomatically false, SkipSteps false, UDAEnableTagReadback false, WithAlarmHandling true
   // inherited from GRAPH_BASE
   VAR
      OFF_SQ_BASE : Bool;
   END_VAR
   VAR_INPUT
      OFF_SQ { ExternalWritable := 'False'} : Bool := false;   // Turn sequence off
      INIT_SQ { ExternalWritable := 'False'} : Bool := false;   // Set sequence to initial state
      ACK_EF { ExternalWritable := 'False'} : Bool := false;   // Acknowledge all errors and faults
      S_PREV { ExternalWritable := 'False'} : Bool := false;   // Output previous step in parameter S_NO
      S_NEXT { ExternalWritable := 'False'} : Bool := false;   // Indicate next step in parameter S_NO
      SW_AUTO { ExternalWritable := 'False'} : Bool := false;   // Automatic mode
      SW_TAP { ExternalWritable := 'False'} : Bool := false;   // Semiautomatic/switch with transition
      SW_TOP { ExternalWritable := 'False'} : Bool := false;   // Semiautomatic/ignore transition
      SW_MAN { ExternalWritable := 'False'} : Bool := false;   // Manual mode
      S_SEL { ExternalWritable := 'False'} : Int := 0;   // Select step to be output to S_NO
      S_ON { ExternalWritable := 'False'} : Bool := false;   // Activate step indicated in S_NO
      S_OFF { ExternalWritable := 'False'} : Bool := false;   // Deactivate step indicated S_NO
      T_PUSH { ExternalWritable := 'False'} : Bool := false;   // Enable transition to switch in semi automatic mode
   END_VAR
   VAR_OUTPUT
      S_NO { ExternalWritable := 'False'} : Int := 0;   // Step number
      S_MORE { ExternalWritable := 'False'} : Bool := false;   // More steps are available and can be shown in S_NO
      S_ACTIVE { ExternalWritable := 'False'} : Bool := false;   // Step indicated in S_NO is active
      ERR_FLT { ExternalWritable := 'False'} : Bool := false;   // Interlock or supervision group error
      AUTO_ON { ExternalWritable := 'False'} : Bool := false;   // Automatic mode is active
      TAP_ON { ExternalWritable := 'False'} : Bool := false;   // Semiautomatic mode/step with transition enabled
      TOP_ON { ExternalWritable := 'False'} : Bool := false;   // Semiautomatic mode/ignore transition enabled
      MAN_ON { ExternalWritable := 'False'} : Bool := false;   // Manual mode is active
   END_VAR
BEGIN
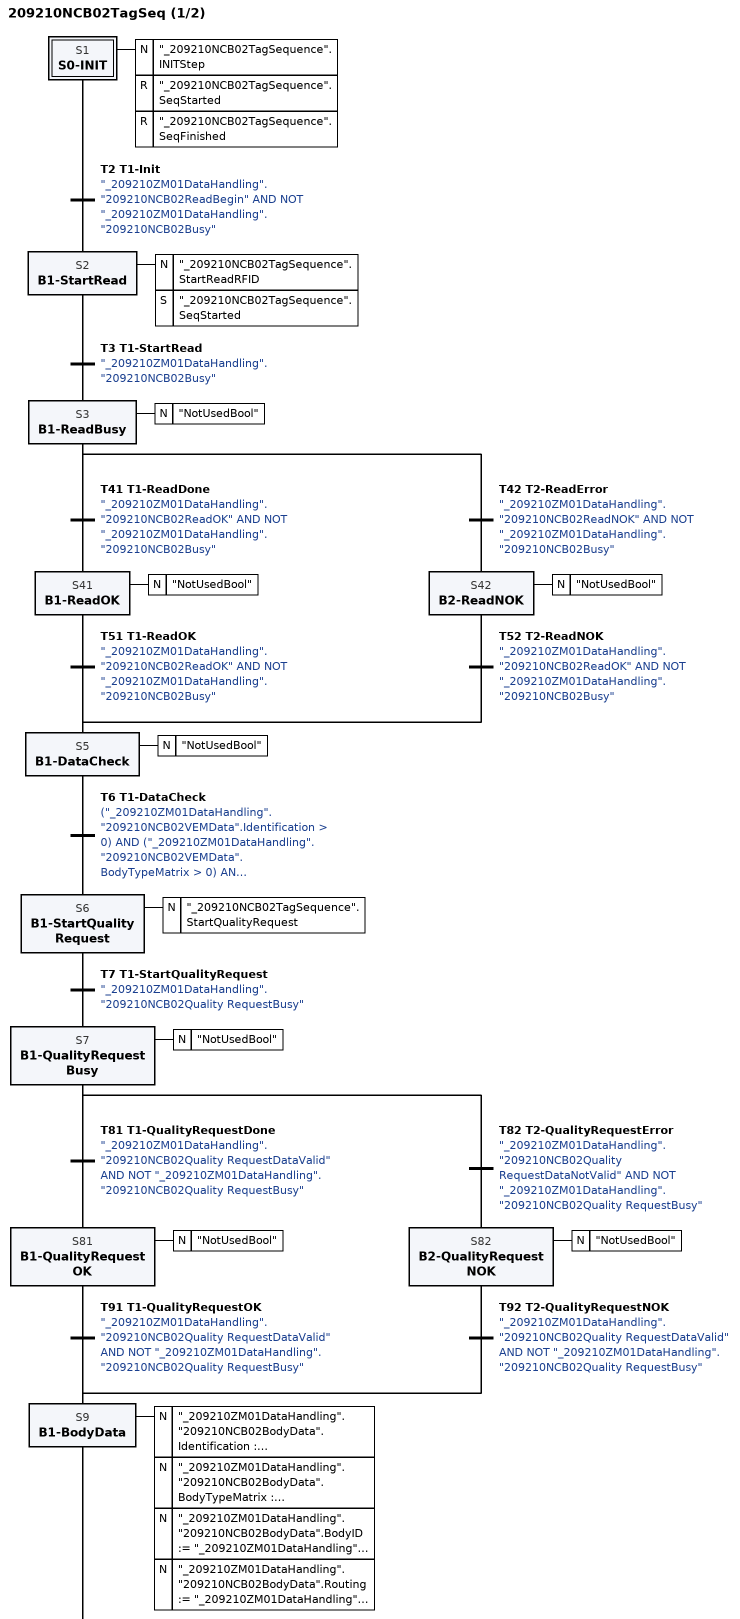
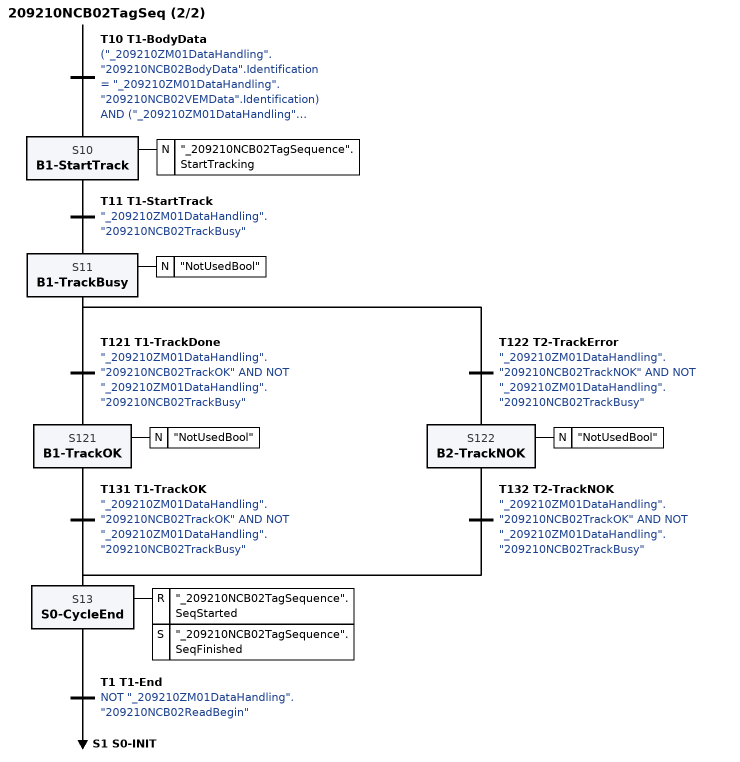
   // sequencer 1: 209210NCB02 Tag Sequence
   // Tag Sequence of 209210NCB02
   INITIAL_STEP "S0-INIT":   // S1, max time T#10S, warning time T#7S
      interlock C := (none);   // Not used
      supervision V := (none);   // Not Used
      // INIT
              N    "_209210NCB02TagSequence".INITStep
              R    "_209210NCB02TagSequence".SeqStarted
              R    "_209210NCB02TagSequence".SeqFinished
   END_STEP
   TRANSITION "T1-Init" FROM "S0-INIT" TO "B1-StartRead"   // T2
      := "_209210ZM01DataHandling"."209210NCB02ReadBegin" AND NOT "_209210ZM01DataHandling"."209210NCB02Busy";
   END_TRANSITION
   STEP "B1-StartRead":   // S2, max time T#10S, warning time T#7S
      interlock C := (none);   // Not Used
      supervision V := (none);   // Not Used
      // Start Getting VEM Data by Reading the Tag with RFID
              N    "_209210NCB02TagSequence".StartReadRFID
              S    "_209210NCB02TagSequence".SeqStarted
   END_STEP
   TRANSITION "T1-StartRead" FROM "B1-StartRead" TO "B1-ReadBusy"   // T3
      := "_209210ZM01DataHandling"."209210NCB02Busy";
   END_TRANSITION
   STEP "B1-ReadBusy":   // S3, max time T#10S, warning time T#7S
      interlock C := (none);   // Not Used
      supervision V := (none);   // Not Used
      // The Tag Reading is Busy
              N    "NotUsedBool"
   END_STEP
   TRANSITION "T1-ReadDone" FROM "B1-ReadBusy" TO "B1-ReadOK"   // T41
      := "_209210ZM01DataHandling"."209210NCB02ReadOK" AND NOT "_209210ZM01DataHandling"."209210NCB02Busy";
   END_TRANSITION
   TRANSITION "T2-ReadError" FROM "B1-ReadBusy" TO "B2-ReadNOK"   // T42
      := "_209210ZM01DataHandling"."209210NCB02ReadNOK" AND NOT "_209210ZM01DataHandling"."209210NCB02Busy";
   END_TRANSITION
   STEP "B2-ReadNOK":   // S42, max time T#10S, warning time T#7S
      interlock C := (none);   // Not Used
      supervision V := (none);   // Not Used
      // Reading of Tag is Not OK
              N    "NotUsedBool"
   END_STEP
   TRANSITION "T2-ReadNOK" FROM "B2-ReadNOK" TO "B1-DataCheck"   // T52
      := "_209210ZM01DataHandling"."209210NCB02ReadOK" AND NOT "_209210ZM01DataHandling"."209210NCB02Busy";
   END_TRANSITION
   STEP "B1-TrackOK":   // S121, max time T#10S, warning time T#7S
      interlock C := (none);   // Not Used
      supervision V := (none);   // Not Used
      // Tracking of the Body is OK
              N    "NotUsedBool"
   END_STEP
   TRANSITION "T1-TrackOK" FROM "B1-TrackOK" TO "S0-CycleEnd"   // T131
      := "_209210ZM01DataHandling"."209210NCB02TrackOK" AND NOT "_209210ZM01DataHandling"."209210NCB02TrackBusy";
   END_TRANSITION
   STEP "B1-ReadOK":   // S41, max time T#10S, warning time T#7S
      interlock C := (none);   // Not Used
      supervision V := (none);   // Not Used
      // Reading of Tag is OK
              N    "NotUsedBool"
   END_STEP
   TRANSITION "T1-ReadOK" FROM "B1-ReadOK" TO "B1-DataCheck"   // T51
      := "_209210ZM01DataHandling"."209210NCB02ReadOK" AND NOT "_209210ZM01DataHandling"."209210NCB02Busy";
   END_TRANSITION
   STEP "S0-CycleEnd":   // S13, max time T#10S, warning time T#7S
      interlock C := (none);   // Not Used
      supervision V := (none);   // Not Used
      // Finished
              R    "_209210NCB02TagSequence".SeqStarted
              S    "_209210NCB02TagSequence".SeqFinished
   END_STEP
   TRANSITION "T1-End" FROM "S0-CycleEnd" TO "S0-INIT"   // T1, jump
      := NOT "_209210ZM01DataHandling"."209210NCB02ReadBegin";
   END_TRANSITION
   STEP "B1-DataCheck":   // S5, max time T#10S, warning time T#7S
      interlock C := (none);   // Not Used
      supervision V := (none);   // Not Used
      // Check if the Received Data is Valid
              N    "NotUsedBool"
   END_STEP
   TRANSITION "T1-DataCheck" FROM "B1-DataCheck" TO "B1-StartQualityRequest"   // T6
      := ("_209210ZM01DataHandling"."209210NCB02VEMData".Identification > 0) AND ("_209210ZM01DataHandling"."209210NCB02VEMData".BodyTypeMatrix > 0) AND ("_209210ZM01DataHandling"."209210NCB02VEMData".BodyID > 0) AND ("_209210ZM01DataHandling"."209210NCB02VEMData".BodyID <= 9999999) AND "_209210ZM01DataHandling"."209210NCB02VEMDataValid";
   END_TRANSITION
   STEP "B1-StartTrack":   // S10, max time T#10S, warning time T#7S
      interlock C := (none);   // Not Used
      supervision V := (none);   // Not Used
      // Start Tracking the Body
              N    "_209210NCB02TagSequence".StartTracking
   END_STEP
   TRANSITION "T1-StartTrack" FROM "B1-StartTrack" TO "B1-TrackBusy"   // T11
      := "_209210ZM01DataHandling"."209210NCB02TrackBusy";
   END_TRANSITION
   STEP "B2-TrackNOK":   // S122, max time T#10S, warning time T#7S
      interlock C := (none);   // Not Used
      supervision V := (none);   // Not Used
      // Tracking of the Body is Not OK
              N    "NotUsedBool"
   END_STEP
   TRANSITION "T2-TrackNOK" FROM "B2-TrackNOK" TO "S0-CycleEnd"   // T132
      := "_209210ZM01DataHandling"."209210NCB02TrackOK" AND NOT "_209210ZM01DataHandling"."209210NCB02TrackBusy";
   END_TRANSITION
   STEP "B1-BodyData":   // S9, max time T#10S, warning time T#7S
      interlock C := (none);   // Not Used
      supervision V := (none);   // Not Used
      // Prepare Data for local use (ex. Shift Register)
              N    "_209210ZM01DataHandling"."209210NCB02BodyData".Identification := "_209210ZM01DataHandling"."209210NCB02VEMData".Identification
              N    "_209210ZM01DataHandling"."209210NCB02BodyData".BodyTypeMatrix := "_209210ZM01DataHandling"."209210NCB02VEMData".BodyTypeMatrix
              N    "_209210ZM01DataHandling"."209210NCB02BodyData".BodyID := "_209210ZM01DataHandling"."209210NCB02VEMData".BodyID
              N    "_209210ZM01DataHandling"."209210NCB02BodyData".Routing := "_209210ZM01DataHandling"."209210NCB02Quality RequestVEMData".Routing
   END_STEP
   TRANSITION "T1-BodyData" FROM "B1-BodyData" TO "B1-StartTrack"   // T10
      := ("_209210ZM01DataHandling"."209210NCB02BodyData".Identification = "_209210ZM01DataHandling"."209210NCB02VEMData".Identification) AND ("_209210ZM01DataHandling"."209210NCB02BodyData".BodyTypeMatrix = "_209210ZM01DataHandling"."209210NCB02VEMData".BodyTypeMatrix) AND ("_209210ZM01DataHandling"."209210NCB02BodyData".BodyID = "_209210ZM01DataHandling"."209210NCB02VEMData".BodyID) AND ("_209210ZM01DataHandling"."209210NCB02BodyData".Routing = "_209210ZM01DataHandling"."209210NCB02Quality RequestVEMData".Routing);
   END_TRANSITION
   STEP "B1-TrackBusy":   // S11, max time T#10S, warning time T#7S
      interlock C := (none);   // Not Used
      supervision V := (none);   // Not Used
      // The Body Tracking is Busy
              N    "NotUsedBool"
   END_STEP
   TRANSITION "T1-TrackDone" FROM "B1-TrackBusy" TO "B1-TrackOK"   // T121
      := "_209210ZM01DataHandling"."209210NCB02TrackOK" AND NOT "_209210ZM01DataHandling"."209210NCB02TrackBusy";
   END_TRANSITION
   TRANSITION "T2-TrackError" FROM "B1-TrackBusy" TO "B2-TrackNOK"   // T122
      := "_209210ZM01DataHandling"."209210NCB02TrackNOK" AND NOT "_209210ZM01DataHandling"."209210NCB02TrackBusy";
   END_TRANSITION
   STEP "B1-StartQualityRequest":   // S6, max time T#10S, warning time T#7S
      interlock C := (none);   // Not Used
      supervision V := (none);   // Not Used
      // Start Tracking the Body
              N    "_209210NCB02TagSequence".StartQualityRequest
   END_STEP
   TRANSITION "T1-StartQualityRequest" FROM "B1-StartQualityRequest" TO "B1-QualityRequestBusy"   // T7
      := "_209210ZM01DataHandling"."209210NCB02Quality RequestBusy";
   END_TRANSITION
   STEP "B1-QualityRequestOK":   // S81, max time T#10S, warning time T#7S
      interlock C := (none);   // Not Used
      supervision V := (none);   // Not Used
      // Tracking of the Body is OK
              N    "NotUsedBool"
   END_STEP
   TRANSITION "T1-QualityRequestOK" FROM "B1-QualityRequestOK" TO "B1-BodyData"   // T91
      := "_209210ZM01DataHandling"."209210NCB02Quality RequestDataValid" AND NOT "_209210ZM01DataHandling"."209210NCB02Quality RequestBusy";
   END_TRANSITION
   STEP "B2-QualityRequestNOK":   // S82, max time T#10S, warning time T#7S
      interlock C := (none);   // Not Used
      supervision V := (none);   // Not Used
      // Tracking of the Body is Not OK
              N    "NotUsedBool"
   END_STEP
   TRANSITION "T2-QualityRequestNOK" FROM "B2-QualityRequestNOK" TO "B1-BodyData"   // T92
      := "_209210ZM01DataHandling"."209210NCB02Quality RequestDataValid" AND NOT "_209210ZM01DataHandling"."209210NCB02Quality RequestBusy";
   END_TRANSITION
   STEP "B1-QualityRequestBusy":   // S7, max time T#10S, warning time T#7S
      interlock C := (none);   // Not Used
      supervision V := (none);   // Not Used
      // The Body Tracking is Busy
              N    "NotUsedBool"
   END_STEP
   TRANSITION "T1-QualityRequestDone" FROM "B1-QualityRequestBusy" TO "B1-QualityRequestOK"   // T81
      := "_209210ZM01DataHandling"."209210NCB02Quality RequestDataValid" AND NOT "_209210ZM01DataHandling"."209210NCB02Quality RequestBusy";
   END_TRANSITION
   TRANSITION "T2-QualityRequestError" FROM "B1-QualityRequestBusy" TO "B2-QualityRequestNOK"   // T82
      := "_209210ZM01DataHandling"."209210NCB02Quality RequestDataNotValid" AND NOT "_209210ZM01DataHandling"."209210NCB02Quality RequestBusy";
   END_TRANSITION

   // permanent post-instructions: Not Used
END_FUNCTION_BLOCK

FUNCTION_BLOCK "209220NCB01TagSeq"   // FB390, GRAPH
{ S7_Optimized_Access := 'TRUE' }
VERSION : 0.1
// stored: AcknowledgeErrorsRequired true, AutoNumber false, GraphVersion 6.0, InitialValuesAcquisition false, IsIECCheckEnabled false, LanguageInNetworks FBD, LockOperatingMode false, PermanentILProcessingInMANMode false, SetENOAutomatically false, SkipSteps false, UDAEnableTagReadback false, WithAlarmHandling true
   // inherited from GRAPH_BASE
   VAR
      OFF_SQ_BASE : Bool;
   END_VAR
   VAR_INPUT
      OFF_SQ { ExternalWritable := 'False'} : Bool := false;   // Turn sequence off
      INIT_SQ { ExternalWritable := 'False'} : Bool := false;   // Set sequence to initial state
      ACK_EF { ExternalWritable := 'False'} : Bool := false;   // Acknowledge all errors and faults
      S_PREV { ExternalWritable := 'False'} : Bool := false;   // Output previous step in parameter S_NO
      S_NEXT { ExternalWritable := 'False'} : Bool := false;   // Indicate next step in parameter S_NO
      SW_AUTO { ExternalWritable := 'False'} : Bool := false;   // Automatic mode
      SW_TAP { ExternalWritable := 'False'} : Bool := false;   // Semiautomatic/switch with transition
      SW_TOP { ExternalWritable := 'False'} : Bool := false;   // Semiautomatic/ignore transition
      SW_MAN { ExternalWritable := 'False'} : Bool := false;   // Manual mode
      S_SEL { ExternalWritable := 'False'} : Int := 0;   // Select step to be output to S_NO
      S_ON { ExternalWritable := 'False'} : Bool := false;   // Activate step indicated in S_NO
      S_OFF { ExternalWritable := 'False'} : Bool := false;   // Deactivate step indicated S_NO
      T_PUSH { ExternalWritable := 'False'} : Bool := false;   // Enable transition to switch in semi automatic mode
   END_VAR
   VAR_OUTPUT
      S_NO { ExternalWritable := 'False'} : Int := 0;   // Step number
      S_MORE { ExternalWritable := 'False'} : Bool := false;   // More steps are available and can be shown in S_NO
      S_ACTIVE { ExternalWritable := 'False'} : Bool := false;   // Step indicated in S_NO is active
      ERR_FLT { ExternalWritable := 'False'} : Bool := false;   // Interlock or supervision group error
      AUTO_ON { ExternalWritable := 'False'} : Bool := false;   // Automatic mode is active
      TAP_ON { ExternalWritable := 'False'} : Bool := false;   // Semiautomatic mode/step with transition enabled
      TOP_ON { ExternalWritable := 'False'} : Bool := false;   // Semiautomatic mode/ignore transition enabled
      MAN_ON { ExternalWritable := 'False'} : Bool := false;   // Manual mode is active
   END_VAR
BEGIN
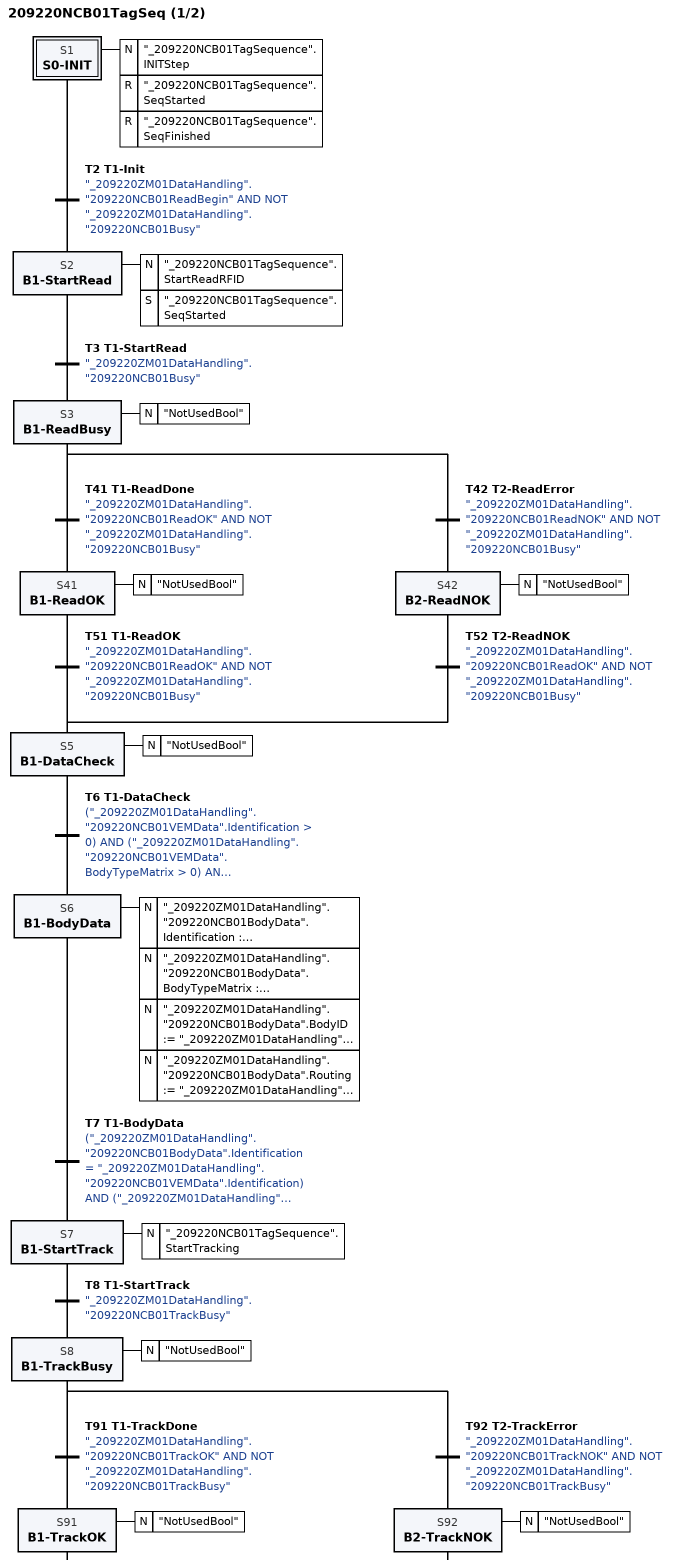
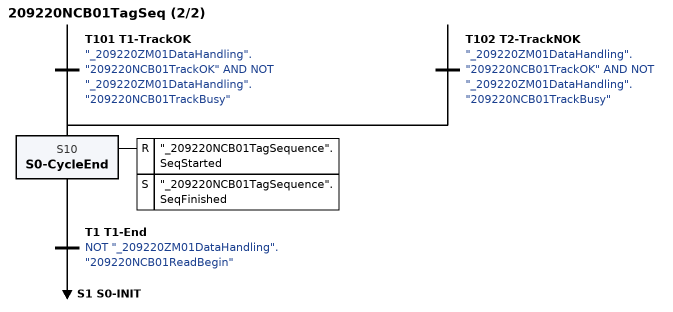
   // sequencer 1: 209220NCB01 Tag Sequence
   // Tag Sequence of 209220NCB01
   INITIAL_STEP "S0-INIT":   // S1, max time T#10S, warning time T#7S
      interlock C := (none);   // Not used
      supervision V := (none);   // Not Used
      // INIT
              N    "_209220NCB01TagSequence".INITStep
              R    "_209220NCB01TagSequence".SeqStarted
              R    "_209220NCB01TagSequence".SeqFinished
   END_STEP
   TRANSITION "T1-Init" FROM "S0-INIT" TO "B1-StartRead"   // T2
      := "_209220ZM01DataHandling"."209220NCB01ReadBegin" AND NOT "_209220ZM01DataHandling"."209220NCB01Busy";
   END_TRANSITION
   STEP "B1-StartRead":   // S2, max time T#10S, warning time T#7S
      interlock C := (none);   // Not Used
      supervision V := (none);   // Not Used
      // Start Getting VEM Data by Reading the Tag with RFID
              N    "_209220NCB01TagSequence".StartReadRFID
              S    "_209220NCB01TagSequence".SeqStarted
   END_STEP
   TRANSITION "T1-StartRead" FROM "B1-StartRead" TO "B1-ReadBusy"   // T3
      := "_209220ZM01DataHandling"."209220NCB01Busy";
   END_TRANSITION
   STEP "B1-ReadBusy":   // S3, max time T#10S, warning time T#7S
      interlock C := (none);   // Not Used
      supervision V := (none);   // Not Used
      // The Tag Reading is Busy
              N    "NotUsedBool"
   END_STEP
   TRANSITION "T1-ReadDone" FROM "B1-ReadBusy" TO "B1-ReadOK"   // T41
      := "_209220ZM01DataHandling"."209220NCB01ReadOK" AND NOT "_209220ZM01DataHandling"."209220NCB01Busy";
   END_TRANSITION
   TRANSITION "T2-ReadError" FROM "B1-ReadBusy" TO "B2-ReadNOK"   // T42
      := "_209220ZM01DataHandling"."209220NCB01ReadNOK" AND NOT "_209220ZM01DataHandling"."209220NCB01Busy";
   END_TRANSITION
   STEP "B1-ReadOK":   // S41, max time T#10S, warning time T#7S
      interlock C := (none);   // Not Used
      supervision V := (none);   // Not Used
      // Reading of Tag is OK
              N    "NotUsedBool"
   END_STEP
   TRANSITION "T1-ReadOK" FROM "B1-ReadOK" TO "B1-DataCheck"   // T51
      := "_209220ZM01DataHandling"."209220NCB01ReadOK" AND NOT "_209220ZM01DataHandling"."209220NCB01Busy";
   END_TRANSITION
   STEP "B2-ReadNOK":   // S42, max time T#10S, warning time T#7S
      interlock C := (none);   // Not Used
      supervision V := (none);   // Not Used
      // Reading of Tag is Not OK
              N    "NotUsedBool"
   END_STEP
   TRANSITION "T2-ReadNOK" FROM "B2-ReadNOK" TO "B1-DataCheck"   // T52
      := "_209220ZM01DataHandling"."209220NCB01ReadOK" AND NOT "_209220ZM01DataHandling"."209220NCB01Busy";
   END_TRANSITION
   STEP "S0-CycleEnd":   // S10, max time T#10S, warning time T#7S
      interlock C := (none);   // Not Used
      supervision V := (none);   // Not Used
      // Finished
              R    "_209220NCB01TagSequence".SeqStarted
              S    "_209220NCB01TagSequence".SeqFinished
   END_STEP
   TRANSITION "T1-End" FROM "S0-CycleEnd" TO "S0-INIT"   // T1, jump
      := NOT "_209220ZM01DataHandling"."209220NCB01ReadBegin";
   END_TRANSITION
   STEP "B1-DataCheck":   // S5, max time T#10S, warning time T#7S
      interlock C := (none);   // Not Used
      supervision V := (none);   // Not Used
      // Check if the Received Data is Valid
              N    "NotUsedBool"
   END_STEP
   TRANSITION "T1-DataCheck" FROM "B1-DataCheck" TO "B1-BodyData"   // T6
      := ("_209220ZM01DataHandling"."209220NCB01VEMData".Identification > 0) AND ("_209220ZM01DataHandling"."209220NCB01VEMData".BodyTypeMatrix > 0) AND ("_209220ZM01DataHandling"."209220NCB01VEMData".BodyID > 0) AND ("_209220ZM01DataHandling"."209220NCB01VEMData".BodyID <= 9999999) AND "_209220ZM01DataHandling"."209220NCB01VEMDataValid";
   END_TRANSITION
   STEP "B1-BodyData":   // S6, max time T#10S, warning time T#7S
      interlock C := (none);   // Not Used
      supervision V := (none);   // Not Used
      // Prepare Data for local use (ex. Shift Register)
              N    "_209220ZM01DataHandling"."209220NCB01BodyData".Identification := "_209220ZM01DataHandling"."209220NCB01VEMData".Identification
              N    "_209220ZM01DataHandling"."209220NCB01BodyData".BodyTypeMatrix := "_209220ZM01DataHandling"."209220NCB01VEMData".BodyTypeMatrix
              N    "_209220ZM01DataHandling"."209220NCB01BodyData".BodyID := "_209220ZM01DataHandling"."209220NCB01VEMData".BodyID
              N    "_209220ZM01DataHandling"."209220NCB01BodyData".Routing := "_209220ZM01DataHandling"."209220NCB01VEMData".Routing
   END_STEP
   TRANSITION "T1-BodyData" FROM "B1-BodyData" TO "B1-StartTrack"   // T7
      := ("_209220ZM01DataHandling"."209220NCB01BodyData".Identification = "_209220ZM01DataHandling"."209220NCB01VEMData".Identification) AND ("_209220ZM01DataHandling"."209220NCB01BodyData".BodyTypeMatrix = "_209220ZM01DataHandling"."209220NCB01VEMData".BodyTypeMatrix) AND ("_209220ZM01DataHandling"."209220NCB01BodyData".BodyID = "_209220ZM01DataHandling"."209220NCB01VEMData".BodyID) AND ("_209220ZM01DataHandling"."209220NCB01BodyData".Routing = "_209220ZM01DataHandling"."209220NCB01VEMData".Routing);
   END_TRANSITION
   STEP "B1-StartTrack":   // S7, max time T#10S, warning time T#7S
      interlock C := (none);   // Not Used
      supervision V := (none);   // Not Used
      // Start Tracking the Body
              N    "_209220NCB01TagSequence".StartTracking
   END_STEP
   TRANSITION "T1-StartTrack" FROM "B1-StartTrack" TO "B1-TrackBusy"   // T8
      := "_209220ZM01DataHandling"."209220NCB01TrackBusy";
   END_TRANSITION
   STEP "B1-TrackOK":   // S91, max time T#10S, warning time T#7S
      interlock C := (none);   // Not Used
      supervision V := (none);   // Not Used
      // Tracking of the Body is OK
              N    "NotUsedBool"
   END_STEP
   TRANSITION "T1-TrackOK" FROM "B1-TrackOK" TO "S0-CycleEnd"   // T101
      := "_209220ZM01DataHandling"."209220NCB01TrackOK" AND NOT "_209220ZM01DataHandling"."209220NCB01TrackBusy";
   END_TRANSITION
   STEP "B2-TrackNOK":   // S92, max time T#10S, warning time T#7S
      interlock C := (none);   // Not Used
      supervision V := (none);   // Not Used
      // Tracking of the Body is Not OK
              N    "NotUsedBool"
   END_STEP
   TRANSITION "T2-TrackNOK" FROM "B2-TrackNOK" TO "S0-CycleEnd"   // T102
      := "_209220ZM01DataHandling"."209220NCB01TrackOK" AND NOT "_209220ZM01DataHandling"."209220NCB01TrackBusy";
   END_TRANSITION
   STEP "B1-TrackBusy":   // S8, max time T#10S, warning time T#7S
      interlock C := (none);   // Not Used
      supervision V := (none);   // Not Used
      // The Body Tracking is Busy
              N    "NotUsedBool"
   END_STEP
   TRANSITION "T1-TrackDone" FROM "B1-TrackBusy" TO "B1-TrackOK"   // T91
      := "_209220ZM01DataHandling"."209220NCB01TrackOK" AND NOT "_209220ZM01DataHandling"."209220NCB01TrackBusy";
   END_TRANSITION
   TRANSITION "T2-TrackError" FROM "B1-TrackBusy" TO "B2-TrackNOK"   // T92
      := "_209220ZM01DataHandling"."209220NCB01TrackNOK" AND NOT "_209220ZM01DataHandling"."209220NCB01TrackBusy";
   END_TRANSITION

   // permanent post-instructions: Not Used
END_FUNCTION_BLOCK

FUNCTION_BLOCK "209220NCB02TagSeq"   // FB391, GRAPH
{ S7_Optimized_Access := 'TRUE' }
VERSION : 0.1
// stored: AcknowledgeErrorsRequired true, AutoNumber false, GraphVersion 6.0, InitialValuesAcquisition false, IsIECCheckEnabled false, LanguageInNetworks FBD, LockOperatingMode false, PermanentILProcessingInMANMode false, SetENOAutomatically false, SkipSteps false, UDAEnableTagReadback false, WithAlarmHandling true
   // inherited from GRAPH_BASE
   VAR
      OFF_SQ_BASE : Bool;
   END_VAR
   VAR_INPUT
      OFF_SQ { ExternalWritable := 'False'} : Bool := false;   // Turn sequence off
      INIT_SQ { ExternalWritable := 'False'} : Bool := false;   // Set sequence to initial state
      ACK_EF { ExternalWritable := 'False'} : Bool := false;   // Acknowledge all errors and faults
      S_PREV { ExternalWritable := 'False'} : Bool := false;   // Output previous step in parameter S_NO
      S_NEXT { ExternalWritable := 'False'} : Bool := false;   // Indicate next step in parameter S_NO
      SW_AUTO { ExternalWritable := 'False'} : Bool := false;   // Automatic mode
      SW_TAP { ExternalWritable := 'False'} : Bool := false;   // Semiautomatic/switch with transition
      SW_TOP { ExternalWritable := 'False'} : Bool := false;   // Semiautomatic/ignore transition
      SW_MAN { ExternalWritable := 'False'} : Bool := false;   // Manual mode
      S_SEL { ExternalWritable := 'False'} : Int := 0;   // Select step to be output to S_NO
      S_ON { ExternalWritable := 'False'} : Bool := false;   // Activate step indicated in S_NO
      S_OFF { ExternalWritable := 'False'} : Bool := false;   // Deactivate step indicated S_NO
      T_PUSH { ExternalWritable := 'False'} : Bool := false;   // Enable transition to switch in semi automatic mode
   END_VAR
   VAR_OUTPUT
      S_NO { ExternalWritable := 'False'} : Int := 0;   // Step number
      S_MORE { ExternalWritable := 'False'} : Bool := false;   // More steps are available and can be shown in S_NO
      S_ACTIVE { ExternalWritable := 'False'} : Bool := false;   // Step indicated in S_NO is active
      ERR_FLT { ExternalWritable := 'False'} : Bool := false;   // Interlock or supervision group error
      AUTO_ON { ExternalWritable := 'False'} : Bool := false;   // Automatic mode is active
      TAP_ON { ExternalWritable := 'False'} : Bool := false;   // Semiautomatic mode/step with transition enabled
      TOP_ON { ExternalWritable := 'False'} : Bool := false;   // Semiautomatic mode/ignore transition enabled
      MAN_ON { ExternalWritable := 'False'} : Bool := false;   // Manual mode is active
   END_VAR
BEGIN
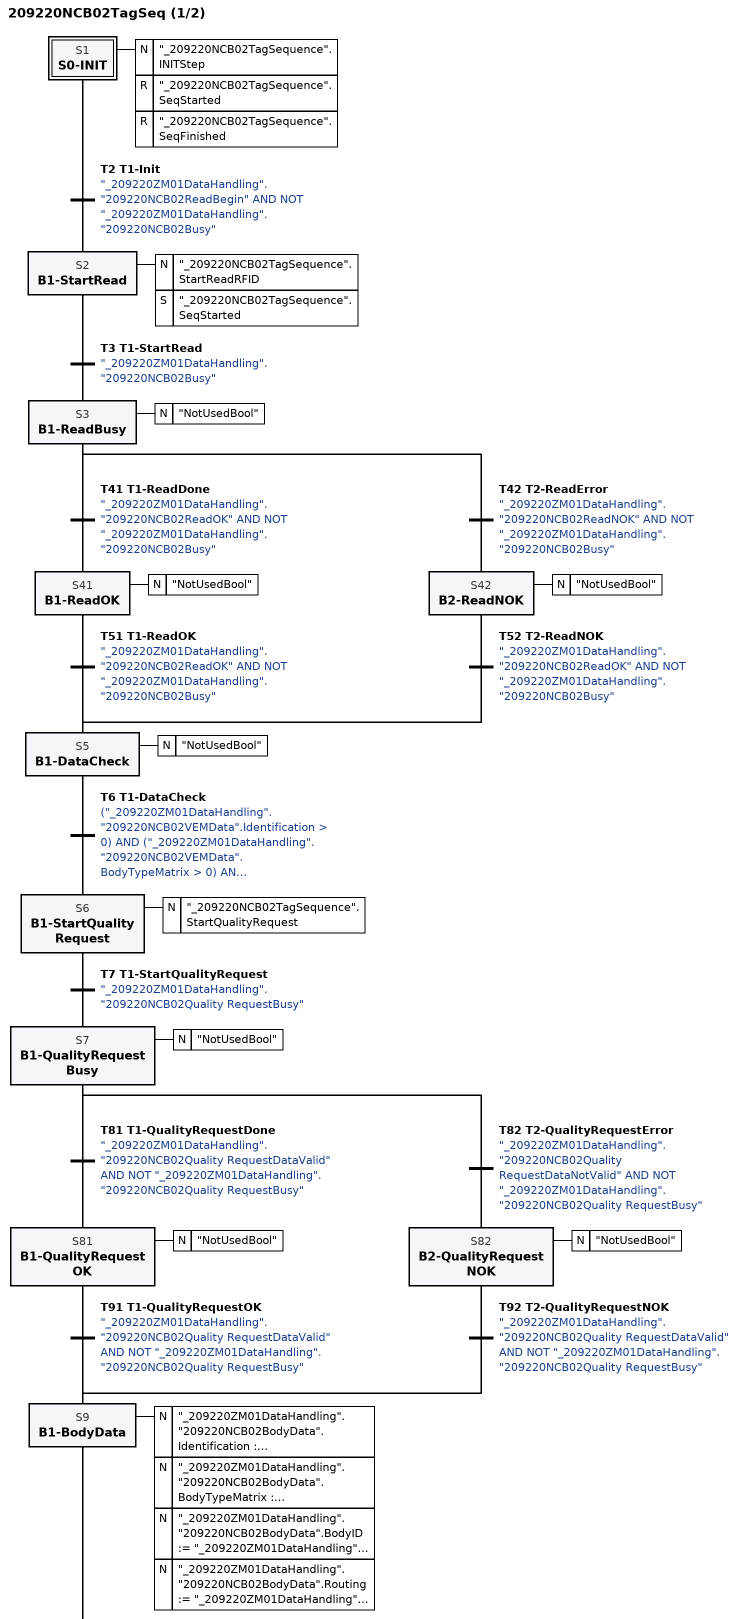
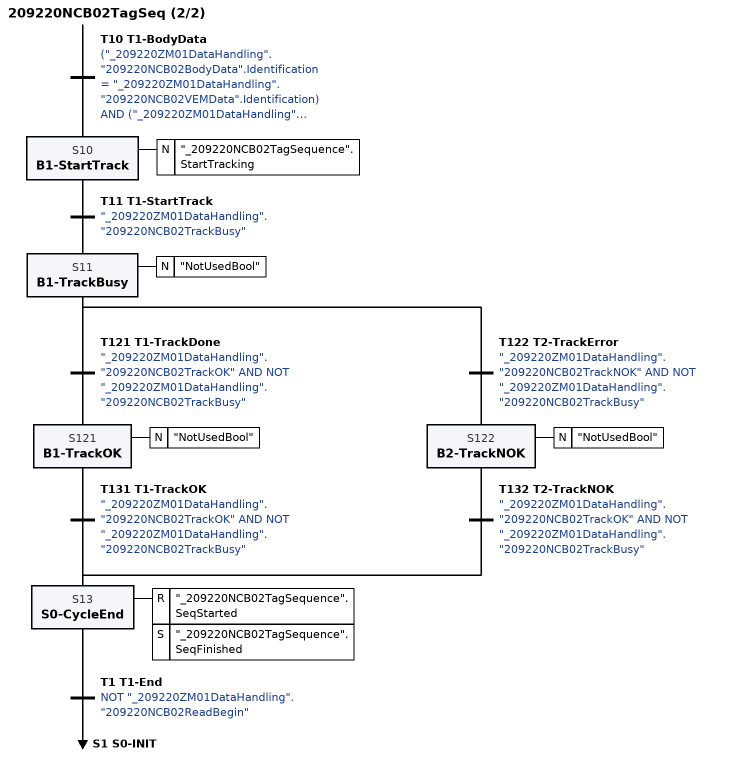
   // sequencer 1: 209220NCB02 Tag Sequence
   // Tag Sequence of 209220NCB02
   INITIAL_STEP "S0-INIT":   // S1, max time T#10S, warning time T#7S
      interlock C := (none);   // Not used
      supervision V := (none);   // Not Used
      // INIT
              N    "_209220NCB02TagSequence".INITStep
              R    "_209220NCB02TagSequence".SeqStarted
              R    "_209220NCB02TagSequence".SeqFinished
   END_STEP
   TRANSITION "T1-Init" FROM "S0-INIT" TO "B1-StartRead"   // T2
      := "_209220ZM01DataHandling"."209220NCB02ReadBegin" AND NOT "_209220ZM01DataHandling"."209220NCB02Busy";
   END_TRANSITION
   STEP "B1-StartRead":   // S2, max time T#10S, warning time T#7S
      interlock C := (none);   // Not Used
      supervision V := (none);   // Not Used
      // Start Getting VEM Data by Reading the Tag with RFID
              N    "_209220NCB02TagSequence".StartReadRFID
              S    "_209220NCB02TagSequence".SeqStarted
   END_STEP
   TRANSITION "T1-StartRead" FROM "B1-StartRead" TO "B1-ReadBusy"   // T3
      := "_209220ZM01DataHandling"."209220NCB02Busy";
   END_TRANSITION
   STEP "B1-ReadBusy":   // S3, max time T#10S, warning time T#7S
      interlock C := (none);   // Not Used
      supervision V := (none);   // Not Used
      // The Tag Reading is Busy
              N    "NotUsedBool"
   END_STEP
   TRANSITION "T1-ReadDone" FROM "B1-ReadBusy" TO "B1-ReadOK"   // T41
      := "_209220ZM01DataHandling"."209220NCB02ReadOK" AND NOT "_209220ZM01DataHandling"."209220NCB02Busy";
   END_TRANSITION
   TRANSITION "T2-ReadError" FROM "B1-ReadBusy" TO "B2-ReadNOK"   // T42
      := "_209220ZM01DataHandling"."209220NCB02ReadNOK" AND NOT "_209220ZM01DataHandling"."209220NCB02Busy";
   END_TRANSITION
   STEP "B1-ReadOK":   // S41, max time T#10S, warning time T#7S
      interlock C := (none);   // Not Used
      supervision V := (none);   // Not Used
      // Reading of Tag is OK
              N    "NotUsedBool"
   END_STEP
   TRANSITION "T1-ReadOK" FROM "B1-ReadOK" TO "B1-DataCheck"   // T51
      := "_209220ZM01DataHandling"."209220NCB02ReadOK" AND NOT "_209220ZM01DataHandling"."209220NCB02Busy";
   END_TRANSITION
   STEP "B2-ReadNOK":   // S42, max time T#10S, warning time T#7S
      interlock C := (none);   // Not Used
      supervision V := (none);   // Not Used
      // Reading of Tag is Not OK
              N    "NotUsedBool"
   END_STEP
   TRANSITION "T2-ReadNOK" FROM "B2-ReadNOK" TO "B1-DataCheck"   // T52
      := "_209220ZM01DataHandling"."209220NCB02ReadOK" AND NOT "_209220ZM01DataHandling"."209220NCB02Busy";
   END_TRANSITION
   STEP "S0-CycleEnd":   // S13, max time T#10S, warning time T#7S
      interlock C := (none);   // Not Used
      supervision V := (none);   // Not Used
      // Finished
              R    "_209220NCB02TagSequence".SeqStarted
              S    "_209220NCB02TagSequence".SeqFinished
   END_STEP
   TRANSITION "T1-End" FROM "S0-CycleEnd" TO "S0-INIT"   // T1, jump
      := NOT "_209220ZM01DataHandling"."209220NCB02ReadBegin";
   END_TRANSITION
   STEP "B1-DataCheck":   // S5, max time T#10S, warning time T#7S
      interlock C := (none);   // Not Used
      supervision V := (none);   // Not Used
      // Check if the Received Data is Valid
              N    "NotUsedBool"
   END_STEP
   TRANSITION "T1-DataCheck" FROM "B1-DataCheck" TO "B1-StartQualityRequest"   // T6
      := ("_209220ZM01DataHandling"."209220NCB02VEMData".Identification > 0) AND ("_209220ZM01DataHandling"."209220NCB02VEMData".BodyTypeMatrix > 0) AND ("_209220ZM01DataHandling"."209220NCB02VEMData".BodyID > 0) AND ("_209220ZM01DataHandling"."209220NCB02VEMData".BodyID <= 9999999) AND "_209220ZM01DataHandling"."209220NCB02VEMDataValid";
   END_TRANSITION
   STEP "B1-BodyData":   // S9, max time T#10S, warning time T#7S
      interlock C := (none);   // Not Used
      supervision V := (none);   // Not Used
      // Prepare Data for local use (ex. Shift Register)
              N    "_209220ZM01DataHandling"."209220NCB02BodyData".Identification := "_209220ZM01DataHandling"."209220NCB02VEMData".Identification
              N    "_209220ZM01DataHandling"."209220NCB02BodyData".BodyTypeMatrix := "_209220ZM01DataHandling"."209220NCB02VEMData".BodyTypeMatrix
              N    "_209220ZM01DataHandling"."209220NCB02BodyData".BodyID := "_209220ZM01DataHandling"."209220NCB02VEMData".BodyID
              N    "_209220ZM01DataHandling"."209220NCB02BodyData".Routing := "_209220ZM01DataHandling"."209220NCB02Quality RequestVEMData".Routing
   END_STEP
   TRANSITION "T1-BodyData" FROM "B1-BodyData" TO "B1-StartTrack"   // T10
      := ("_209220ZM01DataHandling"."209220NCB02BodyData".Identification = "_209220ZM01DataHandling"."209220NCB02VEMData".Identification) AND ("_209220ZM01DataHandling"."209220NCB02BodyData".BodyTypeMatrix = "_209220ZM01DataHandling"."209220NCB02VEMData".BodyTypeMatrix) AND ("_209220ZM01DataHandling"."209220NCB02BodyData".BodyID = "_209220ZM01DataHandling"."209220NCB02VEMData".BodyID) AND ("_209220ZM01DataHandling"."209220NCB02BodyData".Routing = "_209220ZM01DataHandling"."209220NCB02Quality RequestVEMData".Routing);
   END_TRANSITION
   STEP "B1-StartTrack":   // S10, max time T#10S, warning time T#7S
      interlock C := (none);   // Not Used
      supervision V := (none);   // Not Used
      // Start Tracking the Body
              N    "_209220NCB02TagSequence".StartTracking
   END_STEP
   TRANSITION "T1-StartTrack" FROM "B1-StartTrack" TO "B1-TrackBusy"   // T11
      := "_209220ZM01DataHandling"."209220NCB02TrackBusy";
   END_TRANSITION
   STEP "B1-TrackOK":   // S121, max time T#10S, warning time T#7S
      interlock C := (none);   // Not Used
      supervision V := (none);   // Not Used
      // Tracking of the Body is OK
              N    "NotUsedBool"
   END_STEP
   TRANSITION "T1-TrackOK" FROM "B1-TrackOK" TO "S0-CycleEnd"   // T131
      := "_209220ZM01DataHandling"."209220NCB02TrackOK" AND NOT "_209220ZM01DataHandling"."209220NCB02TrackBusy";
   END_TRANSITION
   STEP "B2-TrackNOK":   // S122, max time T#10S, warning time T#7S
      interlock C := (none);   // Not Used
      supervision V := (none);   // Not Used
      // Tracking of the Body is Not OK
              N    "NotUsedBool"
   END_STEP
   TRANSITION "T2-TrackNOK" FROM "B2-TrackNOK" TO "S0-CycleEnd"   // T132
      := "_209220ZM01DataHandling"."209220NCB02TrackOK" AND NOT "_209220ZM01DataHandling"."209220NCB02TrackBusy";
   END_TRANSITION
   STEP "B1-TrackBusy":   // S11, max time T#10S, warning time T#7S
      interlock C := (none);   // Not Used
      supervision V := (none);   // Not Used
      // The Body Tracking is Busy
              N    "NotUsedBool"
   END_STEP
   TRANSITION "T1-TrackDone" FROM "B1-TrackBusy" TO "B1-TrackOK"   // T121
      := "_209220ZM01DataHandling"."209220NCB02TrackOK" AND NOT "_209220ZM01DataHandling"."209220NCB02TrackBusy";
   END_TRANSITION
   TRANSITION "T2-TrackError" FROM "B1-TrackBusy" TO "B2-TrackNOK"   // T122
      := "_209220ZM01DataHandling"."209220NCB02TrackNOK" AND NOT "_209220ZM01DataHandling"."209220NCB02TrackBusy";
   END_TRANSITION
   STEP "B1-StartQualityRequest":   // S6, max time T#10S, warning time T#7S
      interlock C := (none);   // Not Used
      supervision V := (none);   // Not Used
      // Start Tracking the Body
              N    "_209220NCB02TagSequence".StartQualityRequest
   END_STEP
   TRANSITION "T1-StartQualityRequest" FROM "B1-StartQualityRequest" TO "B1-QualityRequestBusy"   // T7
      := "_209220ZM01DataHandling"."209220NCB02Quality RequestBusy";
   END_TRANSITION
   STEP "B1-QualityRequestOK":   // S81, max time T#10S, warning time T#7S
      interlock C := (none);   // Not Used
      supervision V := (none);   // Not Used
      // Tracking of the Body is OK
              N    "NotUsedBool"
   END_STEP
   TRANSITION "T1-QualityRequestOK" FROM "B1-QualityRequestOK" TO "B1-BodyData"   // T91
      := "_209220ZM01DataHandling"."209220NCB02Quality RequestDataValid" AND NOT "_209220ZM01DataHandling"."209220NCB02Quality RequestBusy";
   END_TRANSITION
   STEP "B2-QualityRequestNOK":   // S82, max time T#10S, warning time T#7S
      interlock C := (none);   // Not Used
      supervision V := (none);   // Not Used
      // Tracking of the Body is Not OK
              N    "NotUsedBool"
   END_STEP
   TRANSITION "T2-QualityRequestNOK" FROM "B2-QualityRequestNOK" TO "B1-BodyData"   // T92
      := "_209220ZM01DataHandling"."209220NCB02Quality RequestDataValid" AND NOT "_209220ZM01DataHandling"."209220NCB02Quality RequestBusy";
   END_TRANSITION
   STEP "B1-QualityRequestBusy":   // S7, max time T#10S, warning time T#7S
      interlock C := (none);   // Not Used
      supervision V := (none);   // Not Used
      // The Body Tracking is Busy
              N    "NotUsedBool"
   END_STEP
   TRANSITION "T1-QualityRequestDone" FROM "B1-QualityRequestBusy" TO "B1-QualityRequestOK"   // T81
      := "_209220ZM01DataHandling"."209220NCB02Quality RequestDataValid" AND NOT "_209220ZM01DataHandling"."209220NCB02Quality RequestBusy";
   END_TRANSITION
   TRANSITION "T2-QualityRequestError" FROM "B1-QualityRequestBusy" TO "B2-QualityRequestNOK"   // T82
      := "_209220ZM01DataHandling"."209220NCB02Quality RequestDataNotValid" AND NOT "_209220ZM01DataHandling"."209220NCB02Quality RequestBusy";
   END_TRANSITION

   // permanent post-instructions: Not Used
END_FUNCTION_BLOCK

FUNCTION_BLOCK "209230NCB01TagSeq"   // FB440, GRAPH
{ S7_Optimized_Access := 'TRUE' }
VERSION : 0.1
// stored: AcknowledgeErrorsRequired true, AutoNumber false, GraphVersion 6.0, InitialValuesAcquisition false, IsIECCheckEnabled false, LanguageInNetworks FBD, LockOperatingMode false, PermanentILProcessingInMANMode false, SetENOAutomatically false, SkipSteps false, UDAEnableTagReadback false, WithAlarmHandling true
   // inherited from GRAPH_BASE
   VAR
      OFF_SQ_BASE : Bool;
   END_VAR
   VAR_INPUT
      OFF_SQ { ExternalWritable := 'False'} : Bool := false;   // Turn sequence off
      INIT_SQ { ExternalWritable := 'False'} : Bool := false;   // Set sequence to initial state
      ACK_EF { ExternalWritable := 'False'} : Bool := false;   // Acknowledge all errors and faults
      S_PREV { ExternalWritable := 'False'} : Bool := false;   // Output previous step in parameter S_NO
      S_NEXT { ExternalWritable := 'False'} : Bool := false;   // Indicate next step in parameter S_NO
      SW_AUTO { ExternalWritable := 'False'} : Bool := false;   // Automatic mode
      SW_TAP { ExternalWritable := 'False'} : Bool := false;   // Semiautomatic/switch with transition
      SW_TOP { ExternalWritable := 'False'} : Bool := false;   // Semiautomatic/ignore transition
      SW_MAN { ExternalWritable := 'False'} : Bool := false;   // Manual mode
      S_SEL { ExternalWritable := 'False'} : Int := 0;   // Select step to be output to S_NO
      S_ON { ExternalWritable := 'False'} : Bool := false;   // Activate step indicated in S_NO
      S_OFF { ExternalWritable := 'False'} : Bool := false;   // Deactivate step indicated S_NO
      T_PUSH { ExternalWritable := 'False'} : Bool := false;   // Enable transition to switch in semi automatic mode
   END_VAR
   VAR_OUTPUT
      S_NO { ExternalWritable := 'False'} : Int := 0;   // Step number
      S_MORE { ExternalWritable := 'False'} : Bool := false;   // More steps are available and can be shown in S_NO
      S_ACTIVE { ExternalWritable := 'False'} : Bool := false;   // Step indicated in S_NO is active
      ERR_FLT { ExternalWritable := 'False'} : Bool := false;   // Interlock or supervision group error
      AUTO_ON { ExternalWritable := 'False'} : Bool := false;   // Automatic mode is active
      TAP_ON { ExternalWritable := 'False'} : Bool := false;   // Semiautomatic mode/step with transition enabled
      TOP_ON { ExternalWritable := 'False'} : Bool := false;   // Semiautomatic mode/ignore transition enabled
      MAN_ON { ExternalWritable := 'False'} : Bool := false;   // Manual mode is active
   END_VAR
BEGIN
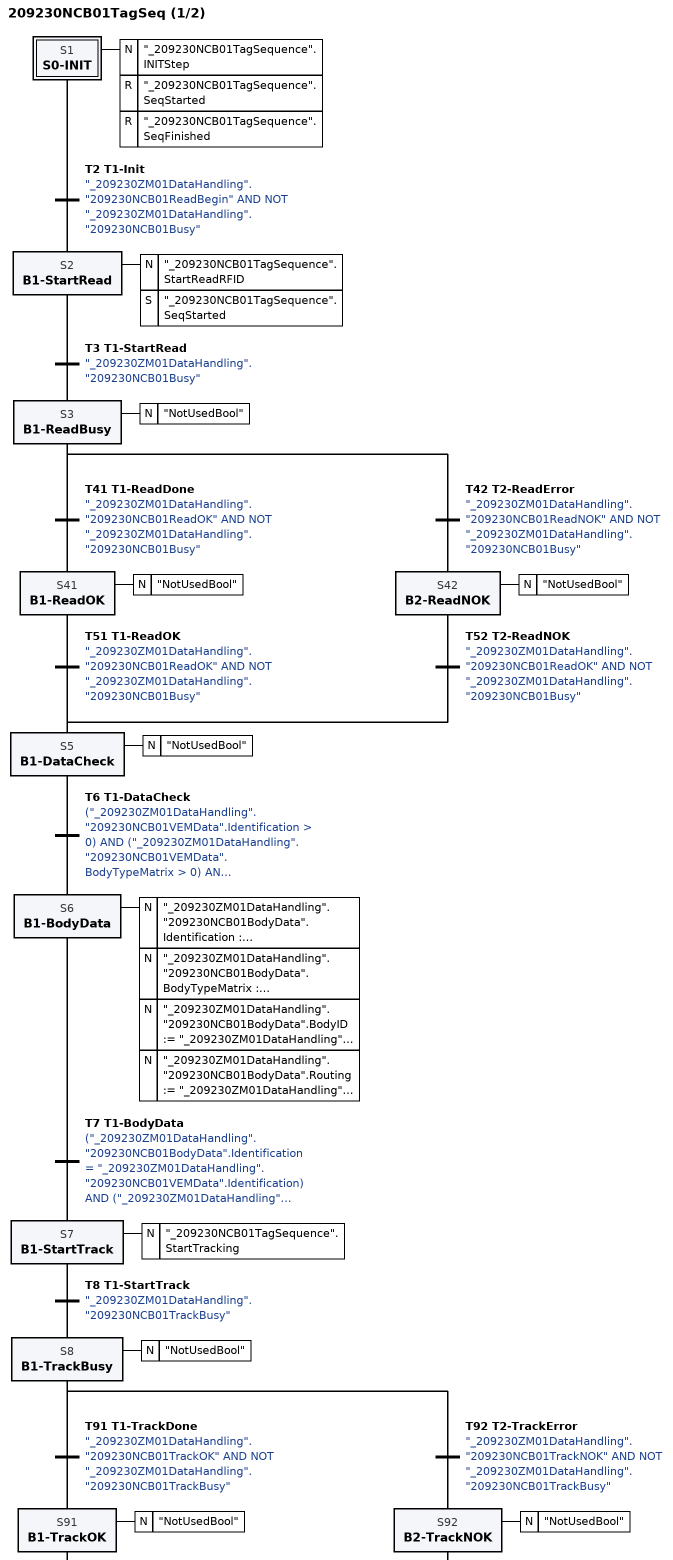
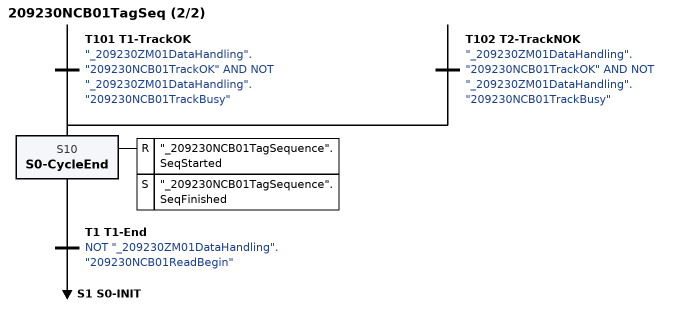
   // sequencer 1: 209230NCB01 Tag Sequence
   // Tag Sequence of 209230NCB01
   INITIAL_STEP "S0-INIT":   // S1, max time T#10S, warning time T#7S
      interlock C := (none);   // Not used
      supervision V := (none);   // Not Used
      // INIT
              N    "_209230NCB01TagSequence".INITStep
              R    "_209230NCB01TagSequence".SeqStarted
              R    "_209230NCB01TagSequence".SeqFinished
   END_STEP
   TRANSITION "T1-Init" FROM "S0-INIT" TO "B1-StartRead"   // T2
      := "_209230ZM01DataHandling"."209230NCB01ReadBegin" AND NOT "_209230ZM01DataHandling"."209230NCB01Busy";
   END_TRANSITION
   STEP "B1-StartRead":   // S2, max time T#10S, warning time T#7S
      interlock C := (none);   // Not Used
      supervision V := (none);   // Not Used
      // Start Getting VEM Data by Reading the Tag with RFID
              N    "_209230NCB01TagSequence".StartReadRFID
              S    "_209230NCB01TagSequence".SeqStarted
   END_STEP
   TRANSITION "T1-StartRead" FROM "B1-StartRead" TO "B1-ReadBusy"   // T3
      := "_209230ZM01DataHandling"."209230NCB01Busy";
   END_TRANSITION
   STEP "B1-ReadBusy":   // S3, max time T#10S, warning time T#7S
      interlock C := (none);   // Not Used
      supervision V := (none);   // Not Used
      // The Tag Reading is Busy
              N    "NotUsedBool"
   END_STEP
   TRANSITION "T1-ReadDone" FROM "B1-ReadBusy" TO "B1-ReadOK"   // T41
      := "_209230ZM01DataHandling"."209230NCB01ReadOK" AND NOT "_209230ZM01DataHandling"."209230NCB01Busy";
   END_TRANSITION
   TRANSITION "T2-ReadError" FROM "B1-ReadBusy" TO "B2-ReadNOK"   // T42
      := "_209230ZM01DataHandling"."209230NCB01ReadNOK" AND NOT "_209230ZM01DataHandling"."209230NCB01Busy";
   END_TRANSITION
   STEP "B1-ReadOK":   // S41, max time T#10S, warning time T#7S
      interlock C := (none);   // Not Used
      supervision V := (none);   // Not Used
      // Reading of Tag is OK
              N    "NotUsedBool"
   END_STEP
   TRANSITION "T1-ReadOK" FROM "B1-ReadOK" TO "B1-DataCheck"   // T51
      := "_209230ZM01DataHandling"."209230NCB01ReadOK" AND NOT "_209230ZM01DataHandling"."209230NCB01Busy";
   END_TRANSITION
   STEP "B2-ReadNOK":   // S42, max time T#10S, warning time T#7S
      interlock C := (none);   // Not Used
      supervision V := (none);   // Not Used
      // Reading of Tag is Not OK
              N    "NotUsedBool"
   END_STEP
   TRANSITION "T2-ReadNOK" FROM "B2-ReadNOK" TO "B1-DataCheck"   // T52
      := "_209230ZM01DataHandling"."209230NCB01ReadOK" AND NOT "_209230ZM01DataHandling"."209230NCB01Busy";
   END_TRANSITION
   STEP "S0-CycleEnd":   // S10, max time T#10S, warning time T#7S
      interlock C := (none);   // Not Used
      supervision V := (none);   // Not Used
      // Finished
              R    "_209230NCB01TagSequence".SeqStarted
              S    "_209230NCB01TagSequence".SeqFinished
   END_STEP
   TRANSITION "T1-End" FROM "S0-CycleEnd" TO "S0-INIT"   // T1, jump
      := NOT "_209230ZM01DataHandling"."209230NCB01ReadBegin";
   END_TRANSITION
   STEP "B1-DataCheck":   // S5, max time T#10S, warning time T#7S
      interlock C := (none);   // Not Used
      supervision V := (none);   // Not Used
      // Check if the Received Data is Valid
              N    "NotUsedBool"
   END_STEP
   TRANSITION "T1-DataCheck" FROM "B1-DataCheck" TO "B1-BodyData"   // T6
      := ("_209230ZM01DataHandling"."209230NCB01VEMData".Identification > 0) AND ("_209230ZM01DataHandling"."209230NCB01VEMData".BodyTypeMatrix > 0) AND ("_209230ZM01DataHandling"."209230NCB01VEMData".BodyID > 0) AND ("_209230ZM01DataHandling"."209230NCB01VEMData".BodyID <= 9999999) AND "_209230ZM01DataHandling"."209230NCB01VEMDataValid";
   END_TRANSITION
   STEP "B1-BodyData":   // S6, max time T#10S, warning time T#7S
      interlock C := (none);   // Not Used
      supervision V := (none);   // Not Used
      // Prepare Data for local use (ex. Shift Register)
              N    "_209230ZM01DataHandling"."209230NCB01BodyData".Identification := "_209230ZM01DataHandling"."209230NCB01VEMData".Identification
              N    "_209230ZM01DataHandling"."209230NCB01BodyData".BodyTypeMatrix := "_209230ZM01DataHandling"."209230NCB01VEMData".BodyTypeMatrix
              N    "_209230ZM01DataHandling"."209230NCB01BodyData".BodyID := "_209230ZM01DataHandling"."209230NCB01VEMData".BodyID
              N    "_209230ZM01DataHandling"."209230NCB01BodyData".Routing := "_209230ZM01DataHandling"."209230NCB01VEMData".Routing
   END_STEP
   TRANSITION "T1-BodyData" FROM "B1-BodyData" TO "B1-StartTrack"   // T7
      := ("_209230ZM01DataHandling"."209230NCB01BodyData".Identification = "_209230ZM01DataHandling"."209230NCB01VEMData".Identification) AND ("_209230ZM01DataHandling"."209230NCB01BodyData".BodyTypeMatrix = "_209230ZM01DataHandling"."209230NCB01VEMData".BodyTypeMatrix) AND ("_209230ZM01DataHandling"."209230NCB01BodyData".BodyID = "_209230ZM01DataHandling"."209230NCB01VEMData".BodyID) AND ("_209230ZM01DataHandling"."209230NCB01BodyData".Routing = "_209230ZM01DataHandling"."209230NCB01VEMData".Routing);
   END_TRANSITION
   STEP "B1-StartTrack":   // S7, max time T#10S, warning time T#7S
      interlock C := (none);   // Not Used
      supervision V := (none);   // Not Used
      // Start Tracking the Body
              N    "_209230NCB01TagSequence".StartTracking
   END_STEP
   TRANSITION "T1-StartTrack" FROM "B1-StartTrack" TO "B1-TrackBusy"   // T8
      := "_209230ZM01DataHandling"."209230NCB01TrackBusy";
   END_TRANSITION
   STEP "B1-TrackOK":   // S91, max time T#10S, warning time T#7S
      interlock C := (none);   // Not Used
      supervision V := (none);   // Not Used
      // Tracking of the Body is OK
              N    "NotUsedBool"
   END_STEP
   TRANSITION "T1-TrackOK" FROM "B1-TrackOK" TO "S0-CycleEnd"   // T101
      := "_209230ZM01DataHandling"."209230NCB01TrackOK" AND NOT "_209230ZM01DataHandling"."209230NCB01TrackBusy";
   END_TRANSITION
   STEP "B2-TrackNOK":   // S92, max time T#10S, warning time T#7S
      interlock C := (none);   // Not Used
      supervision V := (none);   // Not Used
      // Tracking of the Body is Not OK
              N    "NotUsedBool"
   END_STEP
   TRANSITION "T2-TrackNOK" FROM "B2-TrackNOK" TO "S0-CycleEnd"   // T102
      := "_209230ZM01DataHandling"."209230NCB01TrackOK" AND NOT "_209230ZM01DataHandling"."209230NCB01TrackBusy";
   END_TRANSITION
   STEP "B1-TrackBusy":   // S8, max time T#10S, warning time T#7S
      interlock C := (none);   // Not Used
      supervision V := (none);   // Not Used
      // The Body Tracking is Busy
              N    "NotUsedBool"
   END_STEP
   TRANSITION "T1-TrackDone" FROM "B1-TrackBusy" TO "B1-TrackOK"   // T91
      := "_209230ZM01DataHandling"."209230NCB01TrackOK" AND NOT "_209230ZM01DataHandling"."209230NCB01TrackBusy";
   END_TRANSITION
   TRANSITION "T2-TrackError" FROM "B1-TrackBusy" TO "B2-TrackNOK"   // T92
      := "_209230ZM01DataHandling"."209230NCB01TrackNOK" AND NOT "_209230ZM01DataHandling"."209230NCB01TrackBusy";
   END_TRANSITION

   // permanent post-instructions: Not Used
END_FUNCTION_BLOCK

FUNCTION_BLOCK "LGBBeltControl"   // FB6632, FBD
TITLE = LAcofDet / LGBBeltControl
{ S7_Optimized_Access := 'TRUE' }
AUTHOR : VCC
FAMILY : AlarmHandling
NAME : LGBBeltControl
VERSION : 1.0
// ===============================================================================
// This module handles a partdetection with all his functions and alarms
// Functions are DetCheckOn, DetCheckOff and EnableAlarm
// Outputs are DetAlarm and DetSim signal
// ===============================================================================
// ============================================================================
// This module handles Belt Slip Control
// ============================================================================
// stored: AutoNumber false, IsIECCheckEnabled false, IsRetainMemResEnabled false, MemoryReserve 100, SetENOAutomatically False, UDAEnableTagReadback false
   VAR_INPUT
      I_Det1SlipCtrl { ExternalAccessible := 'False'; ExternalVisible := 'False'; ExternalWritable := 'False'} : Bool;   // Actual input from sensor
      I_Det2SlipCtrl { ExternalAccessible := 'False'; ExternalVisible := 'False'; ExternalWritable := 'False'} : Bool;   // Actual input from sensor
      I_MotorRunning { ExternalAccessible := 'False'; ExternalVisible := 'False'; ExternalWritable := 'False'} : Bool;   // Previous detection
      I_EnableAlarm { ExternalAccessible := 'False'; ExternalVisible := 'False'; ExternalWritable := 'False'} : Bool;   // Enable Alarm
      I_AlarmClass { ExternalAccessible := 'False'; ExternalVisible := 'False'; ExternalWritable := 'False'} : Char;   // Alarm class -> A - B - C - D or E
      I_AlarmResetPB { ExternalAccessible := 'False'; ExternalVisible := 'False'; ExternalWritable := 'False'} : Bool;   // Alarm reset pushbutton is activated
   END_VAR
   VAR_OUTPUT
      O_Alarm { ExternalAccessible := 'False'; ExternalVisible := 'False'; ExternalWritable := 'False'} : Bool;   // Detection ON too long alarm / Detection alarm
      O_AlarmABCondition { ExternalAccessible := 'False'; ExternalVisible := 'False'; ExternalWritable := 'False'} : Bool;   // Alarm AB condition
   END_VAR
   VAR_IN_OUT
      H_HMI : "H_HMI";   // H_HMI
      H_BeltControl : "H_GBBeltControl";   // H_KTLBeltSlipControl
      IO_Modes : "Modes";
   END_VAR
   VAR
      CounterSlipCtrl { ExternalAccessible := 'False'; ExternalVisible := 'False'; ExternalWritable := 'False'} : DInt;   // Counter Slip Control
      CounterSlipCtrlL { ExternalAccessible := 'False'; ExternalVisible := 'False'; ExternalWritable := 'False'} : DInt;   // Counter Slip Control Left
      CounterSlipCtrlR { ExternalAccessible := 'False'; ExternalVisible := 'False'; ExternalWritable := 'False'} : DInt;   // Counter Slip Control Right
      AbsCounterSlipCtrl { ExternalAccessible := 'False'; ExternalVisible := 'False'; ExternalWritable := 'False'} : DInt;   // ABS Counter Slip Control
      ResetCount { ExternalAccessible := 'False'; ExternalVisible := 'False'; ExternalWritable := 'False'} : Bool;   // Reset Counters
      AlarmCond { ExternalAccessible := 'False'; ExternalVisible := 'False'; ExternalWritable := 'False'} : Bool;   // Alarm condition / Static variable of O_DetAlarm
      AlarmCondNOCountL { ExternalAccessible := 'False'; ExternalVisible := 'False'; ExternalWritable := 'False'} : Bool;   // Alarm condition / Static variable of O_DetAlarm
      AlarmCondNOCountR { ExternalAccessible := 'False'; ExternalVisible := 'False'; ExternalWritable := 'False'} : Bool;   // Alarm condition / Static variable of O_DetAlarm
      AlarmCondNCCountL { ExternalAccessible := 'False'; ExternalVisible := 'False'; ExternalWritable := 'False'} : Bool;   // Alarm condition / Static variable of O_DetAlarm
      AlarmCondNCCountR { ExternalAccessible := 'False'; ExternalVisible := 'False'; ExternalWritable := 'False'} : Bool;   // Alarm condition / Static variable of O_DetAlarm
      Alarm { ExternalAccessible := 'False'; ExternalVisible := 'False'; ExternalWritable := 'False'} : Bool;   // Alarm / Alarm condition
      AlarmClass_A { ExternalAccessible := 'False'; ExternalVisible := 'False'; ExternalWritable := 'False'} : Bool;   // The alarm is from alarm class A
      AlarmClass_B { ExternalAccessible := 'False'; ExternalVisible := 'False'; ExternalWritable := 'False'} : Bool;   // The alarm is from alarm class B
      AlarmClass_C { ExternalAccessible := 'False'; ExternalVisible := 'False'; ExternalWritable := 'False'} : Bool;   // The alarm is from alarm class C
      AlarmClass_D { ExternalAccessible := 'False'; ExternalVisible := 'False'; ExternalWritable := 'False'} : Bool;   // The alarm is from alarm class D
      AlarmClass_E { ExternalAccessible := 'False'; ExternalVisible := 'False'; ExternalWritable := 'False'} : Bool := false;   // The alarm is from alarm class E
      AlarmFiltered { ExternalAccessible := 'False'; ExternalVisible := 'False'; ExternalWritable := 'False'} : Bool;
      _TimerNoCountL { ExternalAccessible := 'False'; ExternalVisible := 'False'; ExternalWritable := 'False'} : "LTimer";
      _TimerNoCountR { ExternalAccessible := 'False'; ExternalVisible := 'False'; ExternalWritable := 'False'} : "LTimer";
      _TimerNcCountL { ExternalAccessible := 'False'; ExternalVisible := 'False'; ExternalWritable := 'False'} : "LTimer";
      _TimerNcCountR { ExternalAccessible := 'False'; ExternalVisible := 'False'; ExternalWritable := 'False'} : "LTimer";
      _TimerResetCount { ExternalAccessible := 'False'; ExternalVisible := 'False'; ExternalWritable := 'False'} : "LTimer";
      _TimerAlarmFilter { ExternalAccessible := 'False'; ExternalVisible := 'False'; ExternalWritable := 'False'} : "LTimer";
      edge { ExternalAccessible := 'False'; ExternalVisible := 'False'; ExternalWritable := 'False'} : Array[0..1] of Bool;
   END_VAR
   VAR_TEMP   // added for the SCL form of the ladder/FBD networks
      _w1 : Bool;
      _w2 : Bool;
   END_VAR
BEGIN

REGION Network 1: **** 1 - Inputs **** HMI Commands
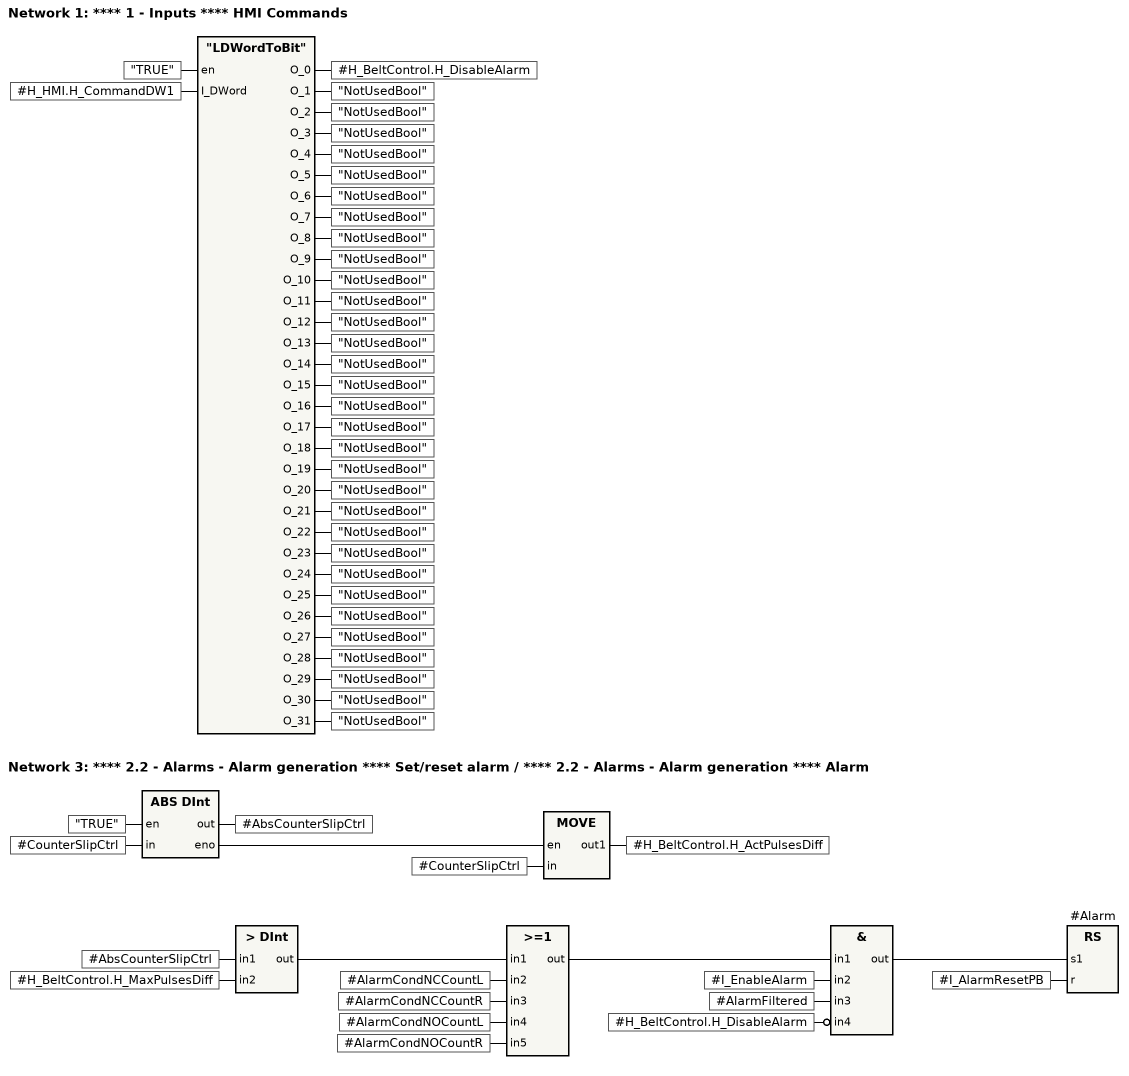
   IF "TRUE" THEN
       "LDWordToBit"(I_DWord := #H_HMI.H_CommandDW1,
                     O_0 => #H_BeltControl.H_DisableAlarm,
                     O_1 => "NotUsedBool",
                     O_2 => "NotUsedBool",
                     O_3 => "NotUsedBool",
                     O_4 => "NotUsedBool",
                     O_5 => "NotUsedBool",
                     O_6 => "NotUsedBool",
                     O_7 => "NotUsedBool",
                     O_8 => "NotUsedBool",
                     O_9 => "NotUsedBool",
                     O_10 => "NotUsedBool",
                     O_11 => "NotUsedBool",
                     O_12 => "NotUsedBool",
                     O_13 => "NotUsedBool",
                     O_14 => "NotUsedBool",
                     O_15 => "NotUsedBool",
                     O_16 => "NotUsedBool",
                     O_17 => "NotUsedBool",
                     O_18 => "NotUsedBool",
                     O_19 => "NotUsedBool",
                     O_20 => "NotUsedBool",
                     O_21 => "NotUsedBool",
                     O_22 => "NotUsedBool",
                     O_23 => "NotUsedBool",
                     O_24 => "NotUsedBool",
                     O_25 => "NotUsedBool",
                     O_26 => "NotUsedBool",
                     O_27 => "NotUsedBool",
                     O_28 => "NotUsedBool",
                     O_29 => "NotUsedBool",
                     O_30 => "NotUsedBool",
                     O_31 => "NotUsedBool");
   END_IF;
END_REGION

NETWORK
TITLE = **** 1 - Inputs **** Alarm class
// Alarm class
// Alarm class = E
      L     #I_AlarmClass;
      L     'E';
      ==I;
      =     #AlarmClass_E;

// Alarm class = D
      L     #I_AlarmClass;
      L     'D';
      ==I;
      =     #AlarmClass_D;

// Alarm class = C
      L     #I_AlarmClass;
      L     'C';
      ==I;
      =     #AlarmClass_C;

// Alarm class = B
      L     #I_AlarmClass;
      L     'B';
      ==I;
      =     #AlarmClass_B;

// Alarm class = A
      AN    #AlarmClass_B;
      AN    #AlarmClass_C;
      AN    #AlarmClass_D;
      AN    #AlarmClass_E;
      =     #AlarmClass_A;


REGION Network 3: **** 2.2 - Alarms - Alarm generation **** Set/reset alarm / **** 2.2 - Alarms - Alarm generation **** Alarm
   // Set/reset alarm
   IF "TRUE" THEN
       #AbsCounterSlipCtrl := ABS(#CounterSlipCtrl);
       #H_BeltControl.H_ActPulsesDiff := #CounterSlipCtrl;
   END_IF;
   IF #I_AlarmResetPB THEN
       #Alarm := FALSE;   // RS flip-flop
   END_IF;
   IF ((#AbsCounterSlipCtrl > #H_BeltControl.H_MaxPulsesDiff) OR #AlarmCondNCCountL OR #AlarmCondNCCountR OR #AlarmCondNOCountL OR #AlarmCondNOCountR) AND #I_EnableAlarm AND #AlarmFiltered AND NOT #H_BeltControl.H_DisableAlarm THEN
       #Alarm := TRUE;
   END_IF;
END_REGION

REGION Network 4: **** 2.2 - Alarms - Alarm generation **** Creating alarm overtime / **** 2.2 - Alarms - Alarm generation **** Pulses counters
   // Creating alarm overtime / Pulses counters
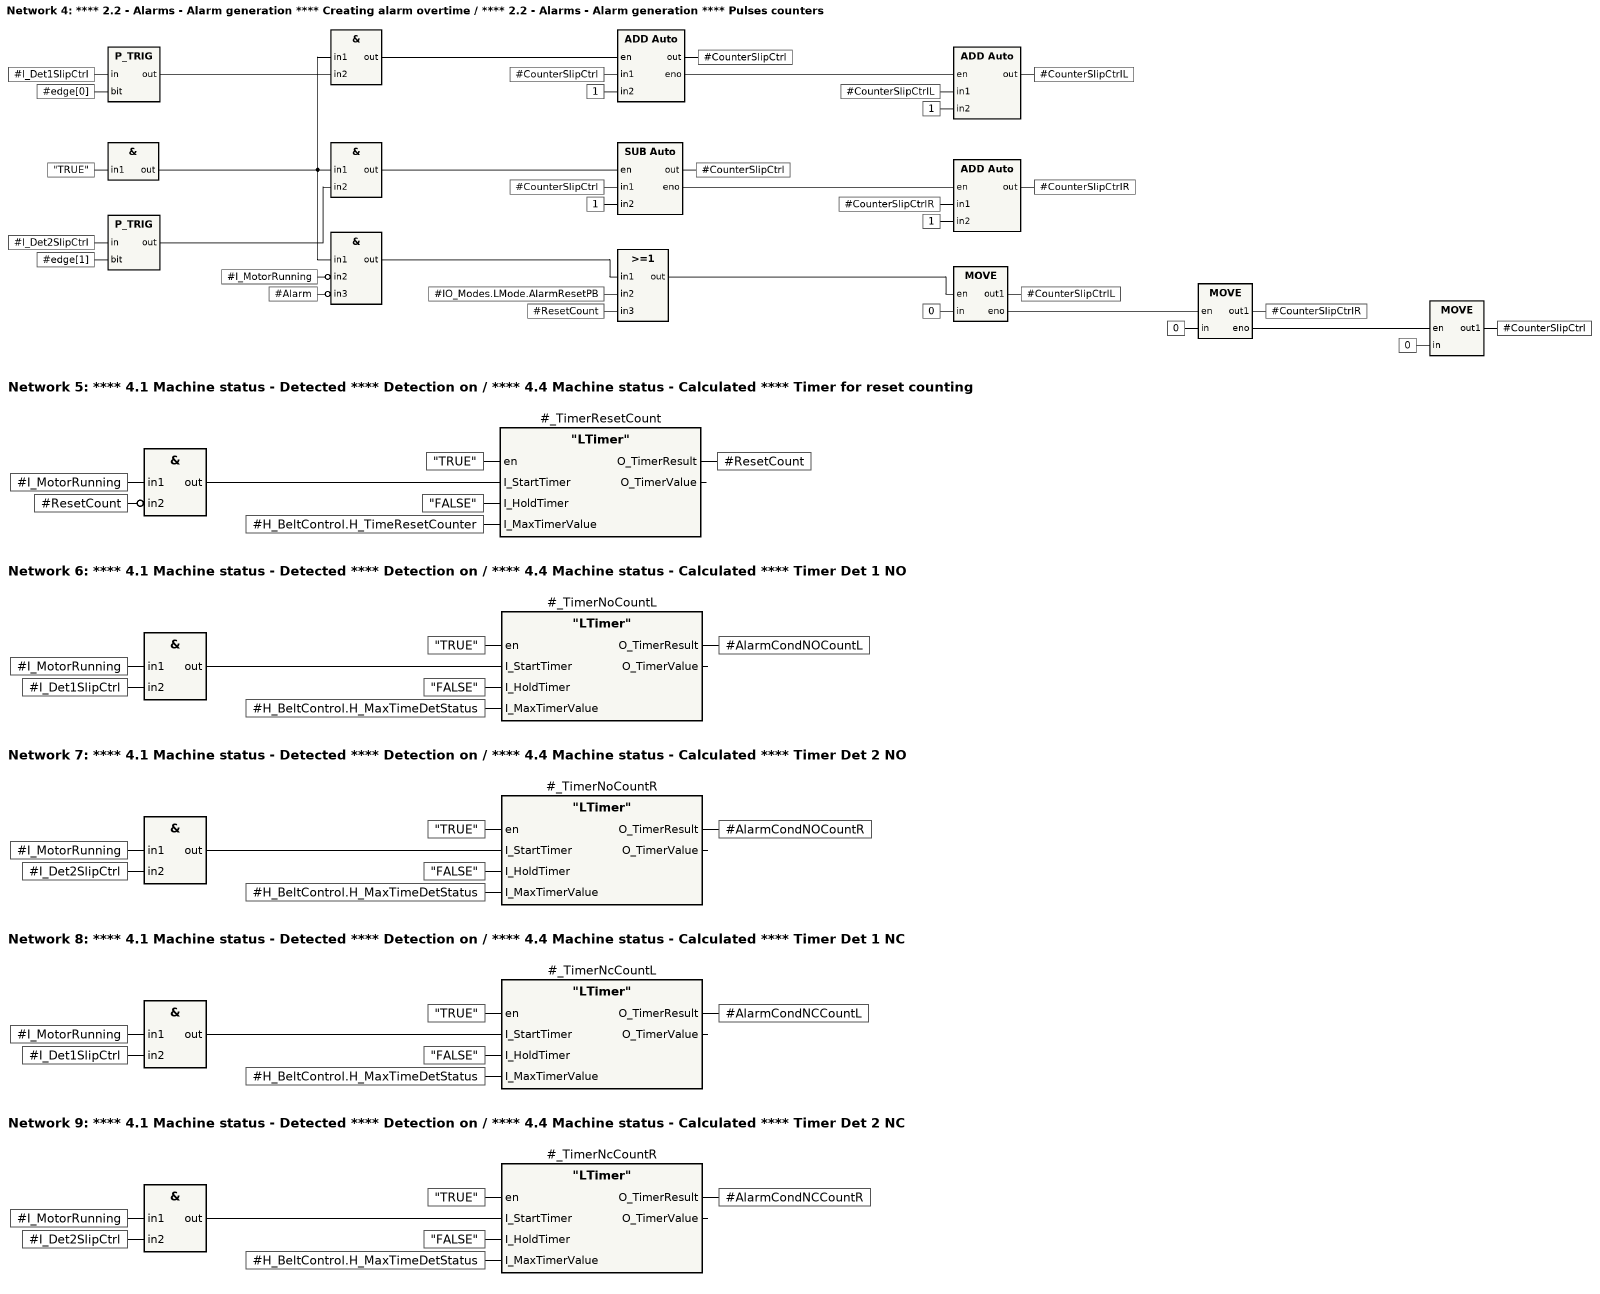
   #_w1 := #I_Det1SlipCtrl AND NOT #edge[0];   // rising edge
   #edge[0] := #I_Det1SlipCtrl;
   IF "TRUE" AND #_w1 THEN
       #CounterSlipCtrl := #CounterSlipCtrl + 1;
       #CounterSlipCtrlL := #CounterSlipCtrlL + 1;
   END_IF;
   #_w2 := #I_Det2SlipCtrl AND NOT #edge[1];   // rising edge
   #edge[1] := #I_Det2SlipCtrl;
   IF "TRUE" AND #_w2 THEN
       #CounterSlipCtrl := #CounterSlipCtrl - 1;
       #CounterSlipCtrlR := #CounterSlipCtrlR + 1;
   END_IF;
   IF ("TRUE" AND NOT #I_MotorRunning AND NOT #Alarm) OR #IO_Modes.LMode.AlarmResetPB OR #ResetCount THEN
       #CounterSlipCtrlL := 0;
       #CounterSlipCtrlR := 0;
       #CounterSlipCtrl := 0;
   END_IF;
END_REGION

REGION Network 5: **** 4.1 Machine status - Detected **** Detection on / **** 4.4 Machine status - Calculated **** Timer for reset counting
   // Detection on / Timer for reset counting
   IF "TRUE" THEN
       #_TimerResetCount(I_StartTimer := #I_MotorRunning AND NOT #ResetCount,   // "LTimer"
                         I_HoldTimer := "FALSE",
                         I_MaxTimerValue := #H_BeltControl.H_TimeResetCounter,
                         O_TimerResult => #ResetCount);
   END_IF;
END_REGION

REGION Network 6: **** 4.1 Machine status - Detected **** Detection on / **** 4.4 Machine status - Calculated **** Timer Det 1 NO
   // Detection on / Timer Det 1 NO
   IF "TRUE" THEN
       #_TimerNoCountL(I_StartTimer := #I_MotorRunning AND #I_Det1SlipCtrl,   // "LTimer"
                       I_HoldTimer := "FALSE",
                       I_MaxTimerValue := #H_BeltControl.H_MaxTimeDetStatus,
                       O_TimerResult => #AlarmCondNOCountL);
   END_IF;
END_REGION

REGION Network 7: **** 4.1 Machine status - Detected **** Detection on / **** 4.4 Machine status - Calculated **** Timer Det 2 NO
   // Detection on / Timer Det 2 NO
   IF "TRUE" THEN
       #_TimerNoCountR(I_StartTimer := #I_MotorRunning AND #I_Det2SlipCtrl,   // "LTimer"
                       I_HoldTimer := "FALSE",
                       I_MaxTimerValue := #H_BeltControl.H_MaxTimeDetStatus,
                       O_TimerResult => #AlarmCondNOCountR);
   END_IF;
END_REGION

REGION Network 8: **** 4.1 Machine status - Detected **** Detection on / **** 4.4 Machine status - Calculated **** Timer Det 1 NC
   // Detection on / Timer Det 1 NC
   IF "TRUE" THEN
       #_TimerNcCountL(I_StartTimer := #I_MotorRunning AND #I_Det1SlipCtrl,   // "LTimer"
                       I_HoldTimer := "FALSE",
                       I_MaxTimerValue := #H_BeltControl.H_MaxTimeDetStatus,
                       O_TimerResult => #AlarmCondNCCountL);
   END_IF;
END_REGION

REGION Network 9: **** 4.1 Machine status - Detected **** Detection on / **** 4.4 Machine status - Calculated **** Timer Det 2 NC
   // Detection on / Timer Det 2 NC
   IF "TRUE" THEN
       #_TimerNcCountR(I_StartTimer := #I_MotorRunning AND #I_Det2SlipCtrl,   // "LTimer"
                       I_HoldTimer := "FALSE",
                       I_MaxTimerValue := #H_BeltControl.H_MaxTimeDetStatus,
                       O_TimerResult => #AlarmCondNCCountR);
   END_IF;
END_REGION

REGION Network 10: **** 4.1 Machine status - Detected **** Detection on / **** 4.4 Machine status - Calculated **** Timer Alarm Filter
   // Detection on / Timer Det 2 NC
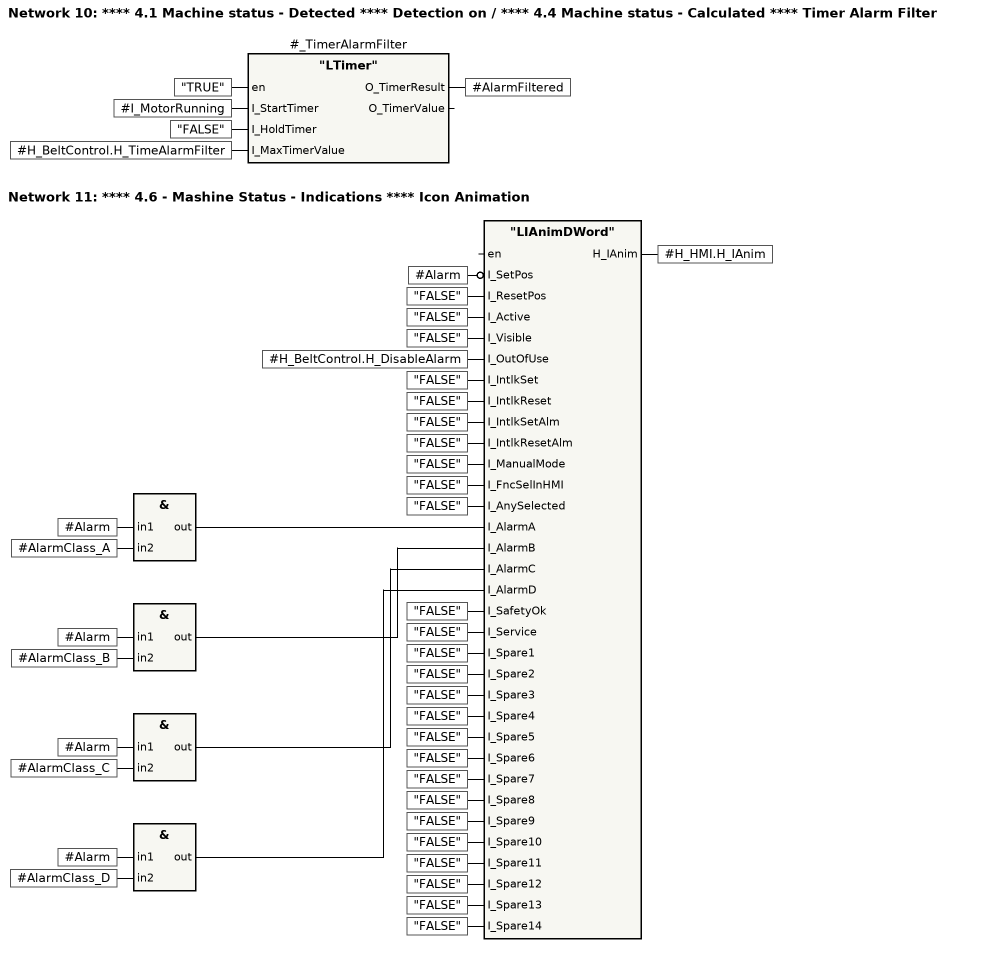
   IF "TRUE" THEN
       #_TimerAlarmFilter(I_StartTimer := #I_MotorRunning,   // "LTimer"
                          I_HoldTimer := "FALSE",
                          I_MaxTimerValue := #H_BeltControl.H_TimeAlarmFilter,
                          O_TimerResult => #AlarmFiltered);
   END_IF;
END_REGION

REGION Network 11: **** 4.6 - Mashine Status - Indications **** Icon Animation
   // Icon Animation
   "LIAnimDWord"(I_SetPos := NOT #Alarm,
                 I_ResetPos := "FALSE",
                 I_Active := "FALSE",
                 I_Visible := "FALSE",
                 I_OutOfUse := #H_BeltControl.H_DisableAlarm,
                 I_IntlkSet := "FALSE",
                 I_IntlkReset := "FALSE",
                 I_IntlkSetAlm := "FALSE",
                 I_IntlkResetAlm := "FALSE",
                 I_ManualMode := "FALSE",
                 I_FncSelInHMI := "FALSE",
                 I_AnySelected := "FALSE",
                 I_AlarmA := #Alarm AND #AlarmClass_A,
                 I_AlarmB := #Alarm AND #AlarmClass_B,
                 I_AlarmC := #Alarm AND #AlarmClass_C,
                 I_AlarmD := #Alarm AND #AlarmClass_D,
                 I_SafetyOk := "FALSE",
                 I_Service := "FALSE",
                 I_Spare1 := "FALSE",
                 I_Spare2 := "FALSE",
                 I_Spare3 := "FALSE",
                 I_Spare4 := "FALSE",
                 I_Spare5 := "FALSE",
                 I_Spare6 := "FALSE",
                 I_Spare7 := "FALSE",
                 I_Spare8 := "FALSE",
                 I_Spare9 := "FALSE",
                 I_Spare10 := "FALSE",
                 I_Spare11 := "FALSE",
                 I_Spare12 := "FALSE",
                 I_Spare13 := "FALSE",
                 I_Spare14 := "FALSE",
                 H_IAnim => #H_HMI.H_IAnim);
END_REGION

REGION Network 12: **** 4.6 - Machine Status - Indications **** Animation
   // Animation
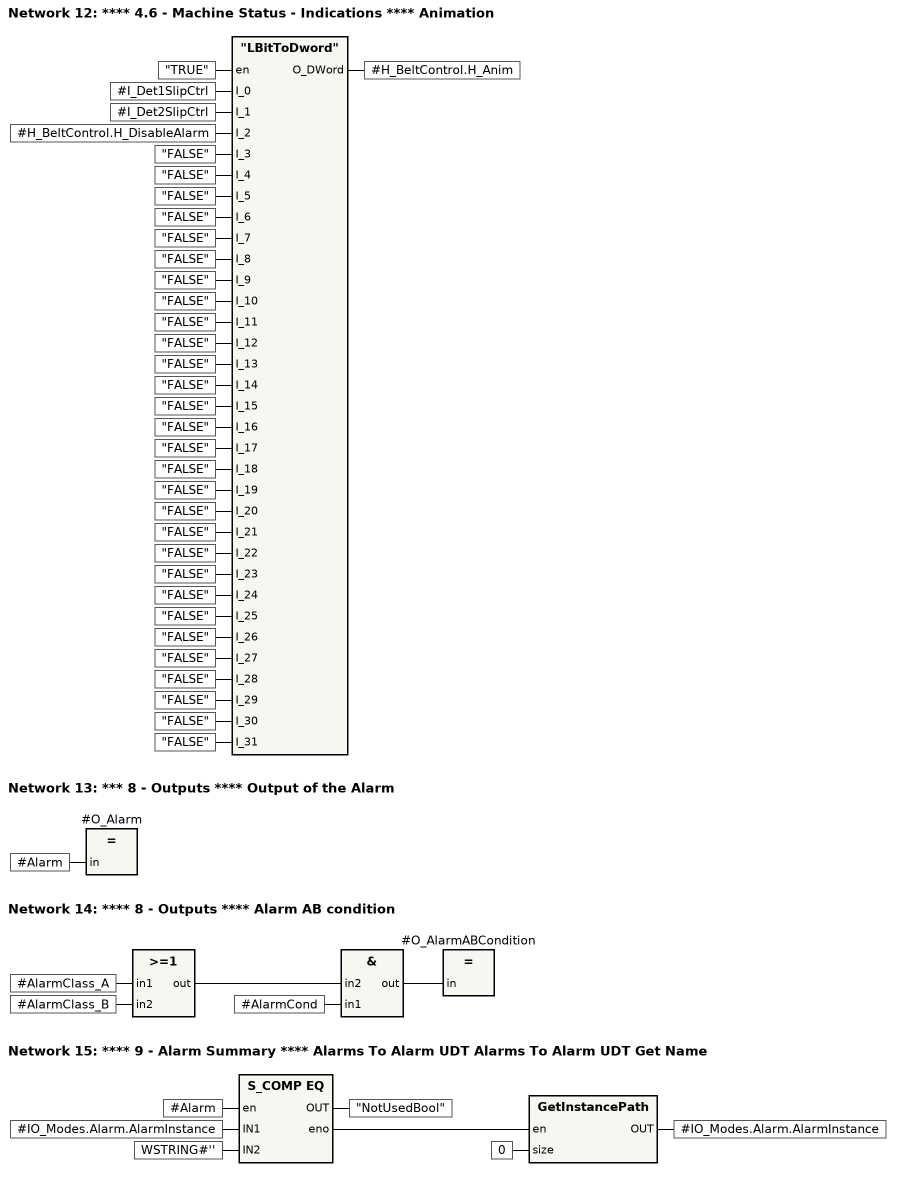
   IF "TRUE" THEN
       "LBitToDword"(I_0 := #I_Det1SlipCtrl,
                     I_1 := #I_Det2SlipCtrl,
                     I_2 := #H_BeltControl.H_DisableAlarm,
                     I_3 := "FALSE",
                     I_4 := "FALSE",
                     I_5 := "FALSE",
                     I_6 := "FALSE",
                     I_7 := "FALSE",
                     I_8 := "FALSE",
                     I_9 := "FALSE",
                     I_10 := "FALSE",
                     I_11 := "FALSE",
                     I_12 := "FALSE",
                     I_13 := "FALSE",
                     I_14 := "FALSE",
                     I_15 := "FALSE",
                     I_16 := "FALSE",
                     I_17 := "FALSE",
                     I_18 := "FALSE",
                     I_19 := "FALSE",
                     I_20 := "FALSE",
                     I_21 := "FALSE",
                     I_22 := "FALSE",
                     I_23 := "FALSE",
                     I_24 := "FALSE",
                     I_25 := "FALSE",
                     I_26 := "FALSE",
                     I_27 := "FALSE",
                     I_28 := "FALSE",
                     I_29 := "FALSE",
                     I_30 := "FALSE",
                     I_31 := "FALSE",
                     O_DWord => #H_BeltControl.H_Anim);
   END_IF;
END_REGION

REGION Network 13: *** 8 - Outputs **** Output of the Alarm
   // Output of the Alarm
   #O_Alarm := #Alarm;
END_REGION

REGION Network 14: **** 8 - Outputs **** Alarm AB condition
   // Alarm AB condition
   #O_AlarmABCondition := (#AlarmClass_A OR #AlarmClass_B) AND #AlarmCond;
END_REGION

REGION Network 15: **** 9 - Alarm Summary **** Alarms To Alarm UDT Alarms To Alarm UDT Get Name
   // Alarm / Alarm D
   S_COMP(EN := #Alarm,
          IN1 := #IO_Modes.Alarm.AlarmInstance,
          IN2 := WSTRING#'',
          OUT => "NotUsedBool",
          ENO => #_w1);
   IF #_w1 THEN GetInstancePath(size := 0, OUT => #IO_Modes.Alarm.AlarmInstance); END_IF;
END_REGION

REGION Network 16: **** 9 - Alarm Summary **** Alarms To Alarm UDT
   // Alarm / Alarm D
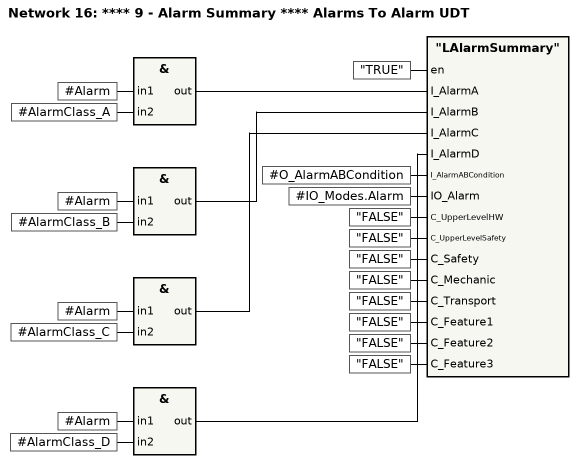
   IF "TRUE" THEN
       "LAlarmSummary"(I_AlarmA := #Alarm AND #AlarmClass_A,
                       I_AlarmB := #Alarm AND #AlarmClass_B,
                       I_AlarmC := #Alarm AND #AlarmClass_C,
                       I_AlarmD := #Alarm AND #AlarmClass_D,
                       I_AlarmABCondition := #O_AlarmABCondition,
                       IO_Alarm := #IO_Modes.Alarm,
                       C_UpperLevelHW := "FALSE",
                       C_UpperLevelSafety := "FALSE",
                       C_Safety := "FALSE",
                       C_Mechanic := "FALSE",
                       C_Transport := "FALSE",
                       C_Feature1 := "FALSE",
                       C_Feature2 := "FALSE",
                       C_Feature3 := "FALSE");
   END_IF;
END_REGION
END_FUNCTION_BLOCK
